LIN {X 0,Y 322.636,Z 898.882,A -85,B 0,C 180,E1 8627.078,E2 8627.078} C_VEL
LIN {X 0,Y 310.386,Z 918.046,A -85,B 0,C 180,E1 8625.849,E2 8625.849} C_VEL
LIN {X 0,Y 296.979,Z 936.905,A -85,B 0,C 180,E1 8624.35,E2 8624.35} C_VEL
LIN {X 0,Y 282.07,Z 955.374,A -85,B 0,C 180,E1 8622.47,E2 8622.47} C_VEL
LIN {X 0,Y 268.359,Z 970.812,A -85,B 0,C 180,E1 8620.504,E2 8620.504} C_VEL
LIN {X 0,Y 251.739,Z 987.693,A -85,B 0,C 180,E1 8617.738,E2 8617.738} C_VEL
LIN {X 0,Y 237.36,Z 1001.003,A -85,B 0,C 180,E1 8614.917,E2 8614.917} C_VEL
LIN {X 0,Y 219.956,Z 1015.757,A -85,B 0,C 180,E1 8610.786,E2 8610.786} C_VEL
LIN {X 0,Y 205.881,Z 1026.76,A -85,B 0,C 180,E1 8606.652,E2 8606.652} C_VEL
LIN {X 0,Y 190.594,Z 1038.003,A -85,B 0,C 180,E1 8600.935,E2 8600.935} C_VEL
LIN {X 0,Y 178.933,Z 1046.164,A -85,B 0,C 180,E1 8595.209,E2 8595.209} C_VEL
LIN {X 0,Y 167.932,Z 1053.856,A -85,B 0,C 180,E1 8587.827,E2 8587.827} C_VEL
LIN {X 0,Y 160.029,Z 1059.461,A -85,B 0,C 180,E1 8579.991,E2 8579.991} C_VEL
LIN {X 0,Y 154.899,Z 1063.661,A -85,B 0,C 180,E1 8571.589,E2 8571.589} C_VEL
LIN {X 0,Y 152.378,Z 1066.343,A -85,B 0,C 180,E1 8562.506,E2 8562.506} C_VEL
LIN {X 0,Y 151.995,Z 1067.325,A -85,B 0,C 180,E1 8555.663,E2 8555.663} C_VEL
LIN {X 0,Y 152.054,Z 1067.454,A -85,B 0,C 180,E1 8550,E2 8550} C_VEL
LIN {X 0,Y 151.999,Z 1066.865,A -85,B 0,C 180,E1 8543.958,E2 8543.958} C_VEL
LIN {X 0,Y 152.481,Z 1065.182,A -85,B 0,C 180,E1 8536.732,E2 8536.732} C_VEL
LIN {X 0,Y 154.529,Z 1062.318,A -85,B 0,C 180,E1 8529.153,E2 8529.153} C_VEL
LIN {X 0,Y 159.895,Z 1057.125,A -85,B 0,C 180,E1 8519.982,E2 8519.982} C_VEL
LIN {X 0,Y 167.312,Z 1050.928,A -85,B 0,C 180,E1 8512.441,E2 8512.441} C_VEL
LIN {X 0,Y 178.116,Z 1042.531,A -85,B 0,C 180,E1 8504.982,E2 8504.982} C_VEL
LIN {X 0,Y 190.201,Z 1032.991,A -85,B 0,C 180,E1 8498.919,E2 8498.919} C_VEL
LIN {X 0,Y 204.082,Z 1021.838,A -85,B 0,C 180,E1 8493.602,E2 8493.602} C_VEL
LIN {X 0,Y 218.709,Z 1009.161,A -85,B 0,C 180,E1 8489.166,E2 8489.166} C_VEL
LIN {X 0,Y 233.696,Z 995.401,A -85,B 0,C 180,E1 8485.474,E2 8485.474} C_VEL
LIN {X 0,Y 248.713,Z 980.22,A -85,B 0,C 180,E1 8482.383,E2 8482.383} C_VEL
LIN {X 0,Y 262.703,Z 964.888,A -85,B 0,C 180,E1 8479.928,E2 8479.928} C_VEL
LIN {X 0,Y 278.275,Z 945.943,A -85,B 0,C 180,E1 8477.567,E2 8477.567} C_VEL
LIN {X 0,Y 290.616,Z 929.27,A -85,B 0,C 180,E1 8475.92,E2 8475.92} C_VEL
LIN {X 0,Y 304.787,Z 907.829,A -85,B 0,C 180,E1 8474.244,E2 8474.244} C_VEL
LIN {X 0,Y 315.652,Z 889.153,A -85,B 0,C 180,E1 8473.081,E2 8473.081} C_VEL
LIN {X 0,Y 326.777,Z 867.511,A -85,B 0,C 180,E1 8471.993,E2 8471.993} C_VEL
LIN {X 0,Y 336.034,Z 846.319,A -85,B 0,C 180,E1 8471.152,E2 8471.152} C_VEL
LIN {X 0,Y 344.895,Z 822.678,A -85,B 0,C 180,E1 8470.416,E2 8470.416} C_VEL
LIN {X 0,Y 351.973,Z 798.939,A -85,B 0,C 180,E1 8469.86,E2 8469.86} C_VEL
LIN {X 0,Y 357.744,Z 774.619,A -85,B 0,C 180,E1 8469.413,E2 8469.413} C_VEL
LIN {X 0,Y 361.712,Z 750.039,A -85,B 0,C 180,E1 8469.033,E2 8469.033} C_VEL
LIN {X 0,Y 375.403,Z 627.088,A -85,B 0,C 180,E1 8467.345,E2 8467.345} C_VEL
LIN {X 0,Y 374.084,Z 623.885,A -85,B 0,C 180,E1 8465.368,E2 8465.368} C_VEL
LIN {X 0,Y 373.134,Z 621.334,A -85,B 0,C 180,E1 8463.38,E2 8463.38} C_VEL
LIN {X 0,Y 372.326,Z 618.216,A -85,B 0,C 180,E1 8458.615,E2 8458.615} C_VEL
LIN {X 0,Y 373.453,Z 622.113,A -85,B 0,C 180,E1 8453.466,E2 8453.466} C_VEL
LIN {X 0,Y 374.948,Z 625.93,A -85,B 0,C 180,E1 8450.87,E2 8450.87} C_VEL
LIN {X 0,Y 375.361,Z 627.187,A -85,B 0,C 180,E1 8450.268,E2 8450.268} C_VEL
LIN {X 0,Y 361.464,Z 750.862,A -85,B 0,C 180,E1 8448.59,E2 8448.59} C_VEL
LIN {X 0,Y 356.777,Z 777.011,A -85,B 0,C 180,E1 8448.155,E2 8448.155} C_VEL
LIN {X 0,Y 351.552,Z 798.416,A -85,B 0,C 180,E1 8447.699,E2 8447.699} C_VEL
LIN {X 0,Y 343.776,Z 823.534,A -85,B 0,C 180,E1 8446.998,E2 8446.998} C_VEL
LIN {X 0,Y 336.067,Z 843.934,A -85,B 0,C 180,E1 8446.27,E2 8446.27} C_VEL
LIN {X 0,Y 326.126,Z 866.42,A -85,B 0,C 180,E1 8445.275,E2 8445.275} C_VEL
LIN {X 0,Y 315.463,Z 886.892,A -85,B 0,C 180,E1 8444.148,E2 8444.148} C_VEL
LIN {X 0,Y 303.574,Z 907.129,A -85,B 0,C 180,E1 8442.781,E2 8442.781} C_VEL
LIN {X 0,Y 290.382,Z 926.631,A -85,B 0,C 180,E1 8441.114,E2 8441.114} C_VEL
LIN {X 0,Y 276.56,Z 945.065,A -85,B 0,C 180,E1 8439.163,E2 8439.163} C_VEL
LIN {X 0,Y 262.07,Z 962.147,A -85,B 0,C 180,E1 8436.853,E2 8436.853} C_VEL
LIN {X 0,Y 248.439,Z 976.868,A -85,B 0,C 180,E1 8434.36,E2 8434.36} C_VEL
LIN {X 0,Y 232.261,Z 992.697,A -85,B 0,C 180,E1 8430.891,E2 8430.891} C_VEL
LIN {X 0,Y 218.488,Z 1005.095,A -85,B 0,C 180,E1 8427.358,E2 8427.358} C_VEL
LIN {X 0,Y 202.958,Z 1018.013,A -85,B 0,C 180,E1 8422.484,E2 8422.484} C_VEL
LIN {X 0,Y 190.742,Z 1027.571,A -85,B 0,C 180,E1 8417.658,E2 8417.658} C_VEL
LIN {X 0,Y 177.939,Z 1037.213,A -85,B 0,C 180,E1 8411.106,E2 8411.106} C_VEL
LIN {X 0,Y 168.28,Z 1044.346,A -85,B 0,C 180,E1 8404.366,E2 8404.366} C_VEL
LIN {X 0,Y 160.311,Z 1050.558,A -85,B 0,C 180,E1 8396.285,E2 8396.285} C_VEL
LIN {X 0,Y 155.313,Z 1054.813,A -85,B 0,C 180,E1 8388,E2 8388} C_VEL
LIN {X 0,Y 152.896,Z 1057.51,A -85,B 0,C 180,E1 8380.17,E2 8380.17} C_VEL
LIN {X 0,Y 152.112,Z 1059.078,A -85,B 0,C 180,E1 8372.26,E2 8372.26} C_VEL
LIN {X 0,Y 152.062,Z 1059.433,A -85,B 0,C 180,E1 8365.474,E2 8365.474} C_VEL
LIN {X 0,Y 152.585,Z 1058.817,A -85,B 0,C 180,E1 8357.895,E2 8357.895} C_VEL
LIN {X 0,Y 154.442,Z 1057.168,A -85,B 0,C 180,E1 8350.327,E2 8350.327} C_VEL
LIN {X 0,Y 158.647,Z 1054.149,A -85,B 0,C 180,E1 8342.2,E2 8342.2} C_VEL
LIN {X 0,Y 166.393,Z 1048.96,A -85,B 0,C 180,E1 8333.494,E2 8333.494} C_VEL
LIN {X 0,Y 175.285,Z 1043.202,A -85,B 0,C 180,E1 8326.802,E2 8326.802} C_VEL
LIN {X 0,Y 188.413,Z 1034.522,A -85,B 0,C 180,E1 8319.691,E2 8319.691} C_VEL
LIN {X 0,Y 201.002,Z 1025.774,A -85,B 0,C 180,E1 8314.548,E2 8314.548} C_VEL
LIN {X 0,Y 216.974,Z 1013.934,A -85,B 0,C 180,E1 8309.428,E2 8309.428} C_VEL
LIN {X 0,Y 230.992,Z 1002.637,A -85,B 0,C 180,E1 8305.794,E2 8305.794} C_VEL
LIN {X 0,Y 246.815,Z 988.886,A -85,B 0,C 180,E1 8302.384,E2 8302.384} C_VEL
LIN {X 0,Y 262.135,Z 974.029,A -85,B 0,C 180,E1 8299.583,E2 8299.583} C_VEL
LIN {X 0,Y 277.791,Z 957.455,A -85,B 0,C 180,E1 8297.128,E2 8297.128} C_VEL
LIN {X 0,Y 292.122,Z 940.304,A -85,B 0,C 180,E1 8295.15,E2 8295.15} C_VEL
LIN {X 0,Y 305.426,Z 922.738,A -85,B 0,C 180,E1 8293.515,E2 8293.515} C_VEL
LIN {X 0,Y 318.945,Z 902.467,A -85,B 0,C 180,E1 8292.008,E2 8292.008} C_VEL
LIN {X 0,Y 329.913,Z 883.896,A -85,B 0,C 180,E1 8290.897,E2 8290.897} C_VEL
LIN {X 0,Y 341.912,Z 860.439,A -85,B 0,C 180,E1 8289.76,E2 8289.76} C_VEL
LIN {X 0,Y 350.295,Z 841.325,A -85,B 0,C 180,E1 8289.021,E2 8289.021} C_VEL
LIN {X 0,Y 358.98,Z 818.103,A -85,B 0,C 180,E1 8288.288,E2 8288.288} C_VEL
LIN {X 0,Y 365.752,Z 795.493,A -85,B 0,C 180,E1 8287.729,E2 8287.729} C_VEL
LIN {X 0,Y 371.547,Z 771.253,A -85,B 0,C 180,E1 8287.27,E2 8287.27} C_VEL
LIN {X 0,Y 375.564,Z 746.851,A -85,B 0,C 180,E1 8286.912,E2 8286.912} C_VEL
LIN {X 0,Y 388.046,Z 637.82,A -85,B 0,C 180,E1 8285.471,E2 8285.471} C_VEL
LIN {X 0,Y 387.076,Z 635.217,A -85,B 0,C 180,E1 8283.406,E2 8283.406} C_VEL
LIN {X 0,Y 386.369,Z 632.327,A -85,B 0,C 180,E1 8279.11,E2 8279.11} C_VEL
LIN {X 0,Y 387.338,Z 635.859,A -85,B 0,C 180,E1 8274.296,E2 8274.296} C_VEL
LIN {X 0,Y 388.067,Z 638.147,A -85,B 0,C 180,E1 8272.782,E2 8272.782} C_VEL
LIN {X 0,Y 374.709,Z 754.049,A -85,B 0,C 180,E1 8271.265,E2 8271.265} C_VEL
LIN {X 0,Y 372.793,Z 765.718,A -85,B 0,C 180,E1 8271.095,E2 8271.095} C_VEL
LIN {X 0,Y 371.277,Z 773.315,A -85,B 0,C 180,E1 8271.153,E2 8271.153} C_VEL
LIN {X 0,Y 365.77,Z 793.42,A -85,B 0,C 180,E1 8271.797,E2 8271.797} C_VEL
LIN {X 0,Y 363.895,Z 799.825,A -85,B 0,C 180,E1 8271.782,E2 8271.782} C_VEL
LIN {X 0,Y 356.423,Z 823.805,A -85,B 0,C 180,E1 8271.287,E2 8271.287} C_VEL
LIN {X 0,Y 348.041,Z 845.479,A -85,B 0,C 180,E1 8270.695,E2 8270.695} C_VEL
LIN {X 0,Y 338.627,Z 866.422,A -85,B 0,C 180,E1 8269.98,E2 8269.98} C_VEL
LIN {X 0,Y 326.946,Z 888.501,A -85,B 0,C 180,E1 8269.023,E2 8269.023} C_VEL
LIN {X 0,Y 315.383,Z 907.692,A -85,B 0,C 180,E1 8267.978,E2 8267.978} C_VEL
LIN {X 0,Y 300.755,Z 928.939,A -85,B 0,C 180,E1 8266.519,E2 8266.519} C_VEL
LIN {X 0,Y 287.707,Z 945.803,A -85,B 0,C 180,E1 8265.05,E2 8265.05} C_VEL
LIN {X 0,Y 270.941,Z 965.149,A -85,B 0,C 180,E1 8262.906,E2 8262.906} C_VEL
LIN {X 0,Y 256.316,Z 980.279,A -85,B 0,C 180,E1 8260.742,E2 8260.742} C_VEL
LIN {X 0,Y 238.838,Z 996.651,A -85,B 0,C 180,E1 8257.7,E2 8257.7} C_VEL
LIN {X 0,Y 223.7,Z 1009.49,A -85,B 0,C 180,E1 8254.541,E2 8254.541} C_VEL
LIN {X 0,Y 207.161,Z 1022.449,A -85,B 0,C 180,E1 8250.319,E2 8250.319} C_VEL
LIN {X 0,Y 192.57,Z 1032.93,A -85,B 0,C 180,E1 8245.648,E2 8245.648} C_VEL
LIN {X 0,Y 178.251,Z 1042.757,A -85,B 0,C 180,E1 8239.719,E2 8239.719} C_VEL
LIN {X 0,Y 166.033,Z 1050.649,A -85,B 0,C 180,E1 8232.884,E2 8232.884} C_VEL
LIN {X 0,Y 156.312,Z 1057.058,A -85,B 0,C 180,E1 8225.149,E2 8225.149} C_VEL
LIN {X 0,Y 148.961,Z 1062.123,A -85,B 0,C 180,E1 8215.912,E2 8215.912} C_VEL
LIN {X 0,Y 145.407,Z 1065.091,A -85,B 0,C 180,E1 8207.612,E2 8207.612} C_VEL
LIN {X 0,Y 144.033,Z 1066.956,A -85,B 0,C 180,E1 8198.383,E2 8198.383} C_VEL
LIN {X 0,Y 144.033,Z 1067.319,A -85,B 0,C 180,E1 8191.482,E2 8191.482} C_VEL
LIN {X 0,Y 144.001,Z 1066.922,A -85,B 0,C 180,E1 8185.22,E2 8185.22} C_VEL
LIN {X 0,Y 144.399,Z 1065.305,A -85,B 0,C 180,E1 8177.198,E2 8177.198} C_VEL
LIN {X 0,Y 146.424,Z 1062.574,A -85,B 0,C 180,E1 8169.201,E2 8169.201} C_VEL
LIN {X 0,Y 151.07,Z 1058.295,A -85,B 0,C 180,E1 8160.674,E2 8160.674} C_VEL
LIN {X 0,Y 159.581,Z 1051.598,A -85,B 0,C 180,E1 8151.662,E2 8151.662} C_VEL
LIN {X 0,Y 169.211,Z 1044.499,A -85,B 0,C 180,E1 8144.839,E2 8144.839} C_VEL
LIN {X 0,Y 183.245,Z 1034.109,A -85,B 0,C 180,E1 8137.702,E2 8137.702} C_VEL
LIN {X 0,Y 196.167,Z 1024.178,A -85,B 0,C 180,E1 8132.751,E2 8132.751} C_VEL
LIN {X 0,Y 213.075,Z 1010.331,A -85,B 0,C 180,E1 8127.683,E2 8127.683} C_VEL
LIN {X 0,Y 227.093,Z 997.928,A -85,B 0,C 180,E1 8124.298,E2 8124.298} C_VEL
LIN {X 0,Y 244.223,Z 981.397,A -85,B 0,C 180,E1 8120.867,E2 8120.867} C_VEL
LIN {X 0,Y 258.302,Z 966.413,A -85,B 0,C 180,E1 8118.487,E2 8118.487} C_VEL
LIN {X 0,Y 273.869,Z 948.18,A -85,B 0,C 180,E1 8116.218,E2 8116.218} C_VEL
LIN {X 0,Y 287.136,Z 930.725,A -85,B 0,C 180,E1 8114.516,E2 8114.516} C_VEL
LIN {X 0,Y 300.657,Z 911.038,A -85,B 0,C 180,E1 8112.986,E2 8112.986} C_VEL
LIN {X 0,Y 312.993,Z 890.336,A -85,B 0,C 180,E1 8111.722,E2 8111.722} C_VEL
LIN {X 0,Y 323.623,Z 870.228,A -85,B 0,C 180,E1 8110.73,E2 8110.73} C_VEL
LIN {X 0,Y 333.881,Z 847.437,A -85,B 0,C 180,E1 8109.846,E2 8109.846} C_VEL
LIN {X 0,Y 341.873,Z 826.674,A -85,B 0,C 180,E1 8109.214,E2 8109.214} C_VEL
LIN {X 0,Y 349.827,Z 801.391,A -85,B 0,C 180,E1 8108.625,E2 8108.625} C_VEL
LIN {X 0,Y 355.241,Z 779.522,A -85,B 0,C 180,E1 8108.229,E2 8108.229} C_VEL
LIN {X 0,Y 360.011,Z 752.727,A -85,B 0,C 180,E1 8107.817,E2 8107.817} C_VEL
LIN {X 0,Y 373.612,Z 633.289,A -85,B 0,C 180,E1 8106.23,E2 8106.23} C_VEL
LIN {X 0,Y 372.089,Z 629.213,A -85,B 0,C 180,E1 8103.235,E2 8103.235} C_VEL
LIN {X 0,Y 371.346,Z 626.202,A -85,B 0,C 180,E1 8098.611,E2 8098.611} C_VEL
LIN {X 0,Y 372.364,Z 629.922,A -85,B 0,C 180,E1 8093.679,E2 8093.679} C_VEL
LIN {X 0,Y 373.577,Z 633.217,A -85,B 0,C 180,E1 8091.404,E2 8091.404} C_VEL
LIN {X 0,Y 360.091,Z 751.213,A -85,B 0,C 180,E1 8089.84,E2 8089.84} C_VEL
LIN {X 0,Y 355.373,Z 777.18,A -85,B 0,C 180,E1 8089.424,E2 8089.424} C_VEL
LIN {X 0,Y 350.07,Z 798.648,A -85,B 0,C 180,E1 8088.985,E2 8088.985} C_VEL
LIN {X 0,Y 342.069,Z 824.119,A -85,B 0,C 180,E1 8088.301,E2 8088.301} C_VEL
LIN {X 0,Y 334.26,Z 844.475,A -85,B 0,C 180,E1 8087.601,E2 8087.601} C_VEL
LIN {X 0,Y 324.182,Z 866.895,A -85,B 0,C 180,E1 8086.645,E2 8086.645} C_VEL
LIN {X 0,Y 313.817,Z 886.539,A -85,B 0,C 180,E1 8085.606,E2 8085.606} C_VEL
LIN {X 0,Y 301.733,Z 906.842,A -85,B 0,C 180,E1 8084.294,E2 8084.294} C_VEL
LIN {X 0,Y 288.501,Z 926.158,A -85,B 0,C 180,E1 8082.713,E2 8082.713} C_VEL
LIN {X 0,Y 275.499,Z 943.251,A -85,B 0,C 180,E1 8080.988,E2 8080.988} C_VEL
LIN {X 0,Y 259.827,Z 961.586,A -85,B 0,C 180,E1 8078.636,E2 8078.636} C_VEL
LIN {X 0,Y 245.843,Z 976.377,A -85,B 0,C 180,E1 8076.222,E2 8076.222} C_VEL
LIN {X 0,Y 229.224,Z 992.292,A -85,B 0,C 180,E1 8072.855,E2 8072.855} C_VEL
LIN {X 0,Y 215.661,Z 1004.157,A -85,B 0,C 180,E1 8069.583,E2 8069.583} C_VEL
LIN {X 0,Y 200.122,Z 1016.792,A -85,B 0,C 180,E1 8065.026,E2 8065.026} C_VEL
LIN {X 0,Y 186.559,Z 1026.959,A -85,B 0,C 180,E1 8060.034,E2 8060.034} C_VEL
LIN {X 0,Y 173.444,Z 1036.446,A -85,B 0,C 180,E1 8053.772,E2 8053.772} C_VEL
LIN {X 0,Y 162.464,Z 1044.017,A -85,B 0,C 180,E1 8046.654,E2 8046.654} C_VEL
LIN {X 0,Y 153.982,Z 1050.121,A -85,B 0,C 180,E1 8038.72,E2 8038.72} C_VEL
LIN {X 0,Y 148.005,Z 1054.743,A -85,B 0,C 180,E1 8029.742,E2 8029.742} C_VEL
LIN {X 0,Y 145.243,Z 1057.412,A -85,B 0,C 180,E1 8021.919,E2 8021.919} C_VEL
LIN {X 0,Y 144.199,Z 1058.976,A -85,B 0,C 180,E1 8014.374,E2 8014.374} C_VEL
LIN {X 0,Y 144.037,Z 1059.569,A -85,B 0,C 180,E1 8007.613,E2 8007.613} C_VEL
LIN {X 0,Y 144.314,Z 1059.398,A -85,B 0,C 180,E1 8000.428,E2 8000.428} C_VEL
LIN {X 0,Y 146.072,Z 1057.914,A -85,B 0,C 180,E1 7991.233,E2 7991.233} C_VEL
LIN {X 0,Y 149.888,Z 1055.271,A -85,B 0,C 180,E1 7983.024,E2 7983.024} C_VEL
LIN {X 0,Y 156.774,Z 1051.046,A -85,B 0,C 180,E1 7974.522,E2 7974.522} C_VEL
LIN {X 0,Y 166.876,Z 1044.865,A -85,B 0,C 180,E1 7966.444,E2 7966.444} C_VEL
LIN {X 0,Y 177.931,Z 1038.053,A -85,B 0,C 180,E1 7960.159,E2 7960.159} C_VEL
LIN {X 0,Y 192.704,Z 1028.454,A -85,B 0,C 180,E1 7953.881,E2 7953.881} C_VEL
LIN {X 0,Y 206.466,Z 1018.863,A -85,B 0,C 180,E1 7949.341,E2 7949.341} C_VEL
LIN {X 0,Y 223.283,Z 1006.192,A -85,B 0,C 180,E1 7944.894,E2 7944.894} C_VEL
LIN {X 0,Y 238.041,Z 993.951,A -85,B 0,C 180,E1 7941.694,E2 7941.694} C_VEL
LIN {X 0,Y 254.411,Z 979.174,A -85,B 0,C 180,E1 7938.705,E2 7938.705} C_VEL
LIN {X 0,Y 269.808,Z 963.547,A -85,B 0,C 180,E1 7936.294,E2 7936.294} C_VEL
LIN {X 0,Y 285.132,Z 946.472,A -85,B 0,C 180,E1 7934.21,E2 7934.21} C_VEL
LIN {X 0,Y 299.537,Z 928.245,A -85,B 0,C 180,E1 7932.472,E2 7932.472} C_VEL
LIN {X 0,Y 312.45,Z 910.056,A -85,B 0,C 180,E1 7931.07,E2 7931.07} C_VEL
LIN {X 0,Y 325.685,Z 888.747,A -85,B 0,C 180,E1 7929.767,E2 7929.767} C_VEL
LIN {X 0,Y 335.946,Z 869.895,A -85,B 0,C 180,E1 7928.831,E2 7928.831} C_VEL
LIN {X 0,Y 346.945,Z 846.423,A -85,B 0,C 180,E1 7927.888,E2 7927.888} C_VEL
LIN {X 0,Y 354.795,Z 826.568,A -85,B 0,C 180,E1 7927.247,E2 7927.247} C_VEL
LIN {X 0,Y 362.673,Z 802.827,A -85,B 0,C 180,E1 7926.638,E2 7926.638} C_VEL
LIN {X 0,Y 368.63,Z 779.656,A -85,B 0,C 180,E1 7926.185,E2 7926.185} C_VEL
LIN {X 0,Y 373.408,Z 755.336,A -85,B 0,C 180,E1 7925.81,E2 7925.81} C_VEL
LIN {X 0,Y 379.555,Z 704.728,A -85,B 0,C 180,E1 7925.156,E2 7925.156} C_VEL
LIN {X 0,Y 386.488,Z 644.435,A -85,B 0,C 180,E1 7924.385,E2 7924.385} C_VEL
LIN {X 0,Y 385.979,Z 642.999,A -85,B 0,C 180,E1 7923.119,E2 7923.119} C_VEL
LIN {X 0,Y 385.387,Z 640.321,A -85,B 0,C 180,E1 7919.108,E2 7919.108} C_VEL
LIN {X 0,Y 386.259,Z 643.666,A -85,B 0,C 180,E1 7914.504,E2 7914.504} C_VEL
LIN {X 0,Y 386.489,Z 644.784,A -85,B 0,C 180,E1 7913.879,E2 7913.879} C_VEL
LIN {X 0,Y 373.686,Z 754.037,A -85,B 0,C 180,E1 7912.483,E2 7912.483} C_VEL
LIN {X 0,Y 368.824,Z 780.191,A -85,B 0,C 180,E1 7912.104,E2 7912.104} C_VEL
LIN {X 0,Y 363.895,Z 799.825,A -85,B 0,C 180,E1 7911.782,E2 7911.782} C_VEL
LIN {X 0,Y 361.669,Z 807.26,A -85,B 0,C 180,E1 7911.819,E2 7911.819} C_VEL
LIN {X 0,Y 354.68,Z 825.951,A -85,B 0,C 180,E1 7912.365,E2 7912.365} C_VEL
LIN {X 0,Y 351.901,Z 833.042,A -85,B 0,C 180,E1 7912.345,E2 7912.345} C_VEL
LIN {X 0,Y 341.59,Z 857.457,A -85,B 0,C 180,E1 7911.643,E2 7911.643} C_VEL
LIN {X 0,Y 331.506,Z 877.698,A -85,B 0,C 180,E1 7910.894,E2 7910.894} C_VEL
LIN {X 0,Y 318.47,Z 900.334,A -85,B 0,C 180,E1 7909.829,E2 7909.829} C_VEL
LIN {X 0,Y 306.359,Z 918.658,A -85,B 0,C 180,E1 7908.744,E2 7908.744} C_VEL
LIN {X 0,Y 292.091,Z 937.956,A -85,B 0,C 180,E1 7907.321,E2 7907.321} C_VEL
LIN {X 0,Y 277.137,Z 955.733,A -85,B 0,C 180,E1 7905.634,E2 7905.634} C_VEL
LIN {X 0,Y 260.71,Z 973.388,A -85,B 0,C 180,E1 7903.499,E2 7903.499} C_VEL
LIN {X 0,Y 244.275,Z 989.022,A -85,B 0,C 180,E1 7901.006,E2 7901.006} C_VEL
LIN {X 0,Y 227.573,Z 1003.58,A -85,B 0,C 180,E1 7897.983,E2 7897.983} C_VEL
LIN {X 0,Y 210.824,Z 1016.635,A -85,B 0,C 180,E1 7894.306,E2 7894.306} C_VEL
LIN {X 0,Y 195.09,Z 1028.025,A -85,B 0,C 180,E1 7890.017,E2 7890.017} C_VEL
LIN {X 0,Y 179.302,Z 1038.497,A -85,B 0,C 180,E1 7884.506,E2 7884.506} C_VEL
LIN {X 0,Y 166.53,Z 1046.54,A -85,B 0,C 180,E1 7878.637,E2 7878.637} C_VEL
LIN {X 0,Y 153.385,Z 1054.528,A -85,B 0,C 180,E1 7870.193,E2 7870.193} C_VEL
LIN {X 0,Y 145.319,Z 1059.505,A -85,B 0,C 180,E1 7862.459,E2 7862.459} C_VEL
LIN {X 0,Y 139.028,Z 1063.816,A -85,B 0,C 180,E1 7852.407,E2 7852.407} C_VEL
LIN {X 0,Y 136.508,Z 1066.001,A -85,B 0,C 180,E1 7843.556,E2 7843.556} C_VEL
LIN {X 0,Y 135.999,Z 1066.928,A -85,B 0,C 180,E1 7835.908,E2 7835.908} C_VEL
LIN {X 0,Y 136.059,Z 1067.021,A -85,B 0,C 180,E1 7830,E2 7830} C_VEL
LIN {X 0,Y 136.006,Z 1066.417,A -85,B 0,C 180,E1 7823.245,E2 7823.245} C_VEL
LIN {X 0,Y 136.711,Z 1064.717,A -85,B 0,C 180,E1 7815.168,E2 7815.168} C_VEL
LIN {X 0,Y 139.354,Z 1061.814,A -85,B 0,C 180,E1 7806.698,E2 7806.698} C_VEL
LIN {X 0,Y 145.833,Z 1056.613,A -85,B 0,C 180,E1 7796.735,E2 7796.735} C_VEL
LIN {X 0,Y 154.501,Z 1050.4,A -85,B 0,C 180,E1 7788.691,E2 7788.691} C_VEL
LIN {X 0,Y 166.227,Z 1042.388,A -85,B 0,C 180,E1 7781.245,E2 7781.245} C_VEL
LIN {X 0,Y 179.96,Z 1032.608,A -85,B 0,C 180,E1 7774.91,E2 7774.91} C_VEL
LIN {X 0,Y 195.382,Z 1021.235,A -85,B 0,C 180,E1 7769.542,E2 7769.542} C_VEL
LIN {X 0,Y 211.129,Z 1008.531,A -85,B 0,C 180,E1 7765.229,E2 7765.229} C_VEL
LIN {X 0,Y 227.067,Z 994.761,A -85,B 0,C 180,E1 7761.699,E2 7761.699} C_VEL
LIN {X 0,Y 243.473,Z 978.966,A -85,B 0,C 180,E1 7758.683,E2 7758.683} C_VEL
LIN {X 0,Y 258.429,Z 963.247,A -85,B 0,C 180,E1 7756.355,E2 7756.355} C_VEL
LIN {X 0,Y 273.92,Z 944.994,A -85,B 0,C 180,E1 7754.268,E2 7754.268} C_VEL
LIN {X 0,Y 287.009,Z 927.872,A -85,B 0,C 180,E1 7752.717,E2 7752.717} C_VEL
LIN {X 0,Y 301.23,Z 906.903,A -85,B 0,C 180,E1 7751.225,E2 7751.225} C_VEL
LIN {X 0,Y 312.372,Z 888.252,A -85,B 0,C 180,E1 7750.168,E2 7750.168} C_VEL
LIN {X 0,Y 324.093,Z 865.864,A -85,B 0,C 180,E1 7749.155,E2 7749.155} C_VEL
LIN {X 0,Y 333.067,Z 845.762,A -85,B 0,C 180,E1 7748.436,E2 7748.436} C_VEL
LIN {X 0,Y 341.865,Z 822.855,A -85,B 0,C 180,E1 7747.787,E2 7747.787} C_VEL
LIN {X 0,Y 349.212,Z 798.836,A -85,B 0,C 180,E1 7747.277,E2 7747.277} C_VEL
LIN {X 0,Y 355.105,Z 774.615,A -85,B 0,C 180,E1 7746.871,E2 7746.871} C_VEL
LIN {X 0,Y 359.227,Z 749.857,A -85,B 0,C 180,E1 7746.514,E2 7746.514} C_VEL
LIN {X 0,Y 371.93,Z 639.67,A -85,B 0,C 180,E1 7745.09,E2 7745.09} C_VEL
LIN {X 0,Y 370.985,Z 636.993,A -85,B 0,C 180,E1 7742.935,E2 7742.935} C_VEL
LIN {X 0,Y 370.365,Z 634.188,A -85,B 0,C 180,E1 7738.608,E2 7738.608} C_VEL
LIN {X 0,Y 371.309,Z 637.843,A -85,B 0,C 180,E1 7733.816,E2 7733.816} C_VEL
LIN {X 0,Y 371.884,Z 639.748,A -85,B 0,C 180,E1 7732.543,E2 7732.543} C_VEL
LIN {X 0,Y 358.891,Z 751.554,A -85,B 0,C 180,E1 7731.1,E2 7731.1} C_VEL
LIN {X 0,Y 354.116,Z 777.471,A -85,B 0,C 180,E1 7730.7,E2 7730.7} C_VEL
LIN {X 0,Y 348.715,Z 799.063,A -85,B 0,C 180,E1 7730.277,E2 7730.277} C_VEL
LIN {X 0,Y 340.54,Z 824.701,A -85,B 0,C 180,E1 7729.616,E2 7729.616} C_VEL
LIN {X 0,Y 332.636,Z 845.015,A -85,B 0,C 180,E1 7728.945,E2 7728.945} C_VEL
LIN {X 0,Y 322.011,Z 868.172,A -85,B 0,C 180,E1 7727.992,E2 7727.992} C_VEL
LIN {X 0,Y 311.508,Z 887.711,A -85,B 0,C 180,E1 7726.993,E2 7726.993} C_VEL
LIN {X 0,Y 299.205,Z 907.957,A -85,B 0,C 180,E1 7725.726,E2 7725.726} C_VEL
LIN {X 0,Y 285.765,Z 927.152,A -85,B 0,C 180,E1 7724.201,E2 7724.201} C_VEL
LIN {X 0,Y 271.231,Z 945.815,A -85,B 0,C 180,E1 7722.355,E2 7722.355} C_VEL
LIN {X 0,Y 256.135,Z 962.851,A -85,B 0,C 180,E1 7720.187,E2 7720.187} C_VEL
LIN {X 0,Y 241.033,Z 978.385,A -85,B 0,C 180,E1 7717.681,E2 7717.681} C_VEL
LIN {X 0,Y 224.836,Z 993.303,A -85,B 0,C 180,E1 7714.526,E2 7714.526} C_VEL
LIN {X 0,Y 210.146,Z 1005.718,A -85,B 0,C 180,E1 7711.102,E2 7711.102} C_VEL
LIN {X 0,Y 193.459,Z 1018.601,A -85,B 0,C 180,E1 7706.318,E2 7706.318} C_VEL
LIN {X 0,Y 180.153,Z 1028.144,A -85,B 0,C 180,E1 7701.498,E2 7701.498} C_VEL
LIN {X 0,Y 165.451,Z 1038.099,A -85,B 0,C 180,E1 7694.51,E2 7694.51} C_VEL
LIN {X 0,Y 155.106,Z 1044.871,A -85,B 0,C 180,E1 7687.764,E2 7687.764} C_VEL
LIN {X 0,Y 145.923,Z 1051.053,A -85,B 0,C 180,E1 7679.111,E2 7679.111} C_VEL
LIN {X 0,Y 140.019,Z 1055.292,A -85,B 0,C 180,E1 7670.046,E2 7670.046} C_VEL
LIN {X 0,Y 137.097,Z 1057.973,A -85,B 0,C 180,E1 7661.357,E2 7661.357} C_VEL
LIN {X 0,Y 136.125,Z 1059.517,A -85,B 0,C 180,E1 7652.526,E2 7652.526} C_VEL
LIN {X 0,Y 136.078,Z 1059.854,A -85,B 0,C 180,E1 7644.941,E2 7644.941} C_VEL
LIN {X 0,Y 136.713,Z 1059.293,A -85,B 0,C 180,E1 7636.895,E2 7636.895} C_VEL
LIN {X 0,Y 138.991,Z 1057.679,A -85,B 0,C 180,E1 7628.476,E2 7628.476} C_VEL
LIN {X 0,Y 143.709,Z 1054.848,A -85,B 0,C 180,E1 7619.937,E2 7619.937} C_VEL
LIN {X 0,Y 152.977,Z 1049.573,A -85,B 0,C 180,E1 7610.167,E2 7610.167} C_VEL
LIN {X 0,Y 163.062,Z 1043.85,A -85,B 0,C 180,E1 7603.138,E2 7603.138} C_VEL
LIN {X 0,Y 177.76,Z 1035.167,A -85,B 0,C 180,E1 7595.803,E2 7595.803} C_VEL
LIN {X 0,Y 191.676,Z 1026.338,A -85,B 0,C 180,E1 7590.601,E2 7590.601} C_VEL
LIN {X 0,Y 208.569,Z 1014.772,A -85,B 0,C 180,E1 7585.673,E2 7585.673} C_VEL
LIN {X 0,Y 224.273,Z 1002.903,A -85,B 0,C 180,E1 7581.994,E2 7581.994} C_VEL
LIN {X 0,Y 240.811,Z 989.282,A -85,B 0,C 180,E1 7578.792,E2 7578.792} C_VEL
LIN {X 0,Y 256.218,Z 975.058,A -85,B 0,C 180,E1 7576.257,E2 7576.257} C_VEL
LIN {X 0,Y 271.177,Z 959.936,A -85,B 0,C 180,E1 7574.131,E2 7574.131} C_VEL
LIN {X 0,Y 286.867,Z 942.134,A -85,B 0,C 180,E1 7572.174,E2 7572.174} C_VEL
LIN {X 0,Y 299.674,Z 925.914,A -85,B 0,C 180,E1 7570.747,E2 7570.747} C_VEL
LIN {X 0,Y 314.092,Z 905.408,A -85,B 0,C 180,E1 7569.298,E2 7569.298} C_VEL
LIN {X 0,Y 325.346,Z 887.102,A -85,B 0,C 180,E1 7568.268,E2 7568.268} C_VEL
LIN {X 0,Y 336.695,Z 866.245,A -85,B 0,C 180,E1 7567.303,E2 7567.303} C_VEL
LIN {X 0,Y 346.692,Z 844.499,A -85,B 0,C 180,E1 7566.502,E2 7566.502} C_VEL
LIN {X 0,Y 354.828,Z 823.837,A -85,B 0,C 180,E1 7565.88,E2 7565.88} C_VEL
LIN {X 0,Y 362.88,Z 798.729,A -85,B 0,C 180,E1 7565.289,E2 7565.289} C_VEL
LIN {X 0,Y 368.398,Z 776.886,A -85,B 0,C 180,E1 7564.897,E2 7564.897} C_VEL
LIN {X 0,Y 373.276,Z 750.254,A -85,B 0,C 180,E1 7564.519,E2 7564.519} C_VEL
LIN {X 0,Y 385.06,Z 651.072,A -85,B 0,C 180,E1 7563.275,E2 7563.275} C_VEL
LIN {X 0,Y 384.406,Z 648.313,A -85,B 0,C 180,E1 7559.106,E2 7559.106} C_VEL
LIN {X 0,Y 385.072,Z 651.262,A -85,B 0,C 180,E1 7554.986,E2 7554.986} C_VEL
LIN {X 0,Y 372.858,Z 753.848,A -85,B 0,C 180,E1 7553.71,E2 7553.71} C_VEL
LIN {X 0,Y 367.945,Z 779.984,A -85,B 0,C 180,E1 7553.346,E2 7553.346} C_VEL
LIN {X 0,Y 362.317,Z 801.977,A -85,B 0,C 180,E1 7553,E2 7553} C_VEL
LIN {X 0,Y 354.003,Z 827.41,A -85,B 0,C 180,E1 7552.484,E2 7552.484} C_VEL
LIN {X 0,Y 351.901,Z 833.042,A -85,B 0,C 180,E1 7552.345,E2 7552.345} C_VEL
LIN {X 0,Y 348.961,Z 840.282,A -85,B 0,C 180,E1 7552.318,E2 7552.318} C_VEL
LIN {X 0,Y 340.298,Z 858.245,A -85,B 0,C 180,E1 7552.791,E2 7552.791} C_VEL
LIN {X 0,Y 336.89,Z 865.112,A -85,B 0,C 180,E1 7552.734,E2 7552.734} C_VEL
LIN {X 0,Y 325.209,Z 886.908,A -85,B 0,C 180,E1 7551.9,E2 7551.9} C_VEL
LIN {X 0,Y 313.827,Z 905.472,A -85,B 0,C 180,E1 7551.003,E2 7551.003} C_VEL
LIN {X 0,Y 299.256,Z 926.414,A -85,B 0,C 180,E1 7549.736,E2 7549.736} C_VEL
LIN {X 0,Y 285.785,Z 943.458,A -85,B 0,C 180,E1 7548.421,E2 7548.421} C_VEL
LIN {X 0,Y 270.221,Z 961.244,A -85,B 0,C 180,E1 7546.697,E2 7546.697} C_VEL
LIN {X 0,Y 254.044,Z 977.534,A -85,B 0,C 180,E1 7544.643,E2 7544.643} C_VEL
LIN {X 0,Y 238.257,Z 992.011,A -85,B 0,C 180,E1 7542.297,E2 7542.297} C_VEL
LIN {X 0,Y 220.432,Z 1006.67,A -85,B 0,C 180,E1 7539.136,E2 7539.136} C_VEL
LIN {X 0,Y 204.985,Z 1018.231,A -85,B 0,C 180,E1 7535.806,E2 7535.806} C_VEL
LIN {X 0,Y 186.511,Z 1030.839,A -85,B 0,C 180,E1 7530.8,E2 7530.8} C_VEL
LIN {X 0,Y 171.931,Z 1039.978,A -85,B 0,C 180,E1 7525.672,E2 7525.672} C_VEL
LIN {X 0,Y 156.524,Z 1049.055,A -85,B 0,C 180,E1 7518.366,E2 7518.366} C_VEL
LIN {X 0,Y 145.248,Z 1055.417,A -85,B 0,C 180,E1 7510.778,E2 7510.778} C_VEL
LIN {X 0,Y 135.786,Z 1060.915,A -85,B 0,C 180,E1 7501.028,E2 7501.028} C_VEL
LIN {X 0,Y 130.572,Z 1064.21,A -85,B 0,C 180,E1 7491.566,E2 7491.566} C_VEL
LIN {X 0,Y 128.359,Z 1066.085,A -85,B 0,C 180,E1 7482.598,E2 7482.598} C_VEL
LIN {X 0,Y 128.002,Z 1066.818,A -85,B 0,C 180,E1 7474.48,E2 7474.48} C_VEL
LIN {X 0,Y 128.037,Z 1066.713,A -85,B 0,C 180,E1 7468.21,E2 7468.21} C_VEL
LIN {X 0,Y 128.044,Z 1065.979,A -85,B 0,C 180,E1 7461.468,E2 7461.468} C_VEL
LIN {X 0,Y 129.155,Z 1064.128,A -85,B 0,C 180,E1 7452.891,E2 7452.891} C_VEL
LIN {X 0,Y 133.454,Z 1060.36,A -85,B 0,C 180,E1 7442.32,E2 7442.32} C_VEL
LIN {X 0,Y 140.894,Z 1055.047,A -85,B 0,C 180,E1 7432.899,E2 7432.899} C_VEL
LIN {X 0,Y 151.918,Z 1047.938,A -85,B 0,C 180,E1 7424.159,E2 7424.159} C_VEL
LIN {X 0,Y 165.139,Z 1039.209,A -85,B 0,C 180,E1 7416.943,E2 7416.943} C_VEL
LIN {X 0,Y 179.785,Z 1029.321,A -85,B 0,C 180,E1 7411.076,E2 7411.076} C_VEL
LIN {X 0,Y 195.964,Z 1017.429,A -85,B 0,C 180,E1 7406.101,E2 7406.101} C_VEL
LIN {X 0,Y 211.756,Z 1004.997,A -85,B 0,C 180,E1 7402.257,E2 7402.257} C_VEL
LIN {X 0,Y 228.856,Z 990.097,A -85,B 0,C 180,E1 7398.863,E2 7398.863} C_VEL
LIN {X 0,Y 243.866,Z 975.771,A -85,B 0,C 180,E1 7396.375,E2 7396.375} C_VEL
LIN {X 0,Y 260.896,Z 957.673,A -85,B 0,C 180,E1 7393.972,E2 7393.972} C_VEL
LIN {X 0,Y 274.295,Z 941.809,A -85,B 0,C 180,E1 7392.328,E2 7392.328} C_VEL
LIN {X 0,Y 289.489,Z 921.719,A -85,B 0,C 180,E1 7390.687,E2 7390.687} C_VEL
LIN {X 0,Y 302.091,Z 902.766,A -85,B 0,C 180,E1 7389.478,E2 7389.478} C_VEL
LIN {X 0,Y 314.82,Z 881.085,A -85,B 0,C 180,E1 7388.372,E2 7388.372} C_VEL
LIN {X 0,Y 325.281,Z 860.292,A -85,B 0,C 180,E1 7387.546,E2 7387.546} C_VEL
LIN {X 0,Y 334.799,Z 838.531,A -85,B 0,C 180,E1 7386.861,E2 7386.861} C_VEL
LIN {X 0,Y 343.033,Z 815.564,A -85,B 0,C 180,E1 7386.299,E2 7386.299} C_VEL
LIN {X 0,Y 349.627,Z 793.272,A -85,B 0,C 180,E1 7385.877,E2 7385.877} C_VEL
LIN {X 0,Y 355.299,Z 767.873,A -85,B 0,C 180,E1 7385.491,E2 7385.491} C_VEL
LIN {X 0,Y 358.865,Z 745.266,A -85,B 0,C 180,E1 7385.182,E2 7385.182} C_VEL
LIN {X 0,Y 370.36,Z 646.203,A -85,B 0,C 180,E1 7383.909,E2 7383.909} C_VEL
LIN {X 0,Y 369.892,Z 644.775,A -85,B 0,C 180,E1 7382.634,E2 7382.634} C_VEL
LIN {X 0,Y 369.384,Z 642.181,A -85,B 0,C 180,E1 7378.604,E2 7378.604} C_VEL
LIN {X 0,Y 370.228,Z 645.651,A -85,B 0,C 180,E1 7374.032,E2 7374.032} C_VEL
LIN {X 0,Y 370.338,Z 646.293,A -85,B 0,C 180,E1 7373.693,E2 7373.693} C_VEL
LIN {X 0,Y 357.88,Z 751.789,A -85,B 0,C 180,E1 7372.369,E2 7372.369} C_VEL
LIN {X 0,Y 353.035,Z 777.762,A -85,B 0,C 180,E1 7371.985,E2 7371.985} C_VEL
LIN {X 0,Y 347.557,Z 799.413,A -85,B 0,C 180,E1 7371.58,E2 7371.58} C_VEL
LIN {X 0,Y 339.664,Z 824.008,A -85,B 0,C 180,E1 7370.979,E2 7370.979} C_VEL
LIN {X 0,Y 331.666,Z 844.431,A -85,B 0,C 180,E1 7370.34,E2 7370.34} C_VEL
LIN {X 0,Y 321.374,Z 866.861,A -85,B 0,C 180,E1 7369.473,E2 7369.473} C_VEL
LIN {X 0,Y 310.217,Z 887.437,A -85,B 0,C 180,E1 7368.479,E2 7368.479} C_VEL
LIN {X 0,Y 297.782,Z 907.691,A -85,B 0,C 180,E1 7367.275,E2 7367.275} C_VEL
LIN {X 0,Y 284.128,Z 926.943,A -85,B 0,C 180,E1 7365.819,E2 7365.819} C_VEL
LIN {X 0,Y 269.735,Z 945.158,A -85,B 0,C 180,E1 7364.104,E2 7364.104} C_VEL
LIN {X 0,Y 254.375,Z 962.289,A -85,B 0,C 180,E1 7362.035,E2 7362.035} C_VEL
LIN {X 0,Y 239.451,Z 977.364,A -85,B 0,C 180,E1 7359.721,E2 7359.721} C_VEL
LIN {X 0,Y 222.273,Z 992.933,A -85,B 0,C 180,E1 7356.59,E2 7356.59} C_VEL
LIN {X 0,Y 207.108,Z 1005.405,A -85,B 0,C 180,E1 7353.272,E2 7353.272} C_VEL
LIN {X 0,Y 189.492,Z 1018.593,A -85,B 0,C 180,E1 7348.507,E2 7348.507} C_VEL
LIN {X 0,Y 175.853,Z 1027.98,A -85,B 0,C 180,E1 7343.843,E2 7343.843} C_VEL
LIN {X 0,Y 160.888,Z 1037.679,A -85,B 0,C 180,E1 7337.168,E2 7337.168} C_VEL
LIN {X 0,Y 149.223,Z 1044.838,A -85,B 0,C 180,E1 7330.035,E2 7330.035} C_VEL
LIN {X 0,Y 139.232,Z 1051.1,A -85,B 0,C 180,E1 7321.136,E2 7321.136} C_VEL
LIN {X 0,Y 132.661,Z 1055.377,A -85,B 0,C 180,E1 7311.674,E2 7311.674} C_VEL
LIN {X 0,Y 129.421,Z 1057.985,A -85,B 0,C 180,E1 7302.947,E2 7302.947} C_VEL
LIN {X 0,Y 128.164,Z 1059.622,A -85,B 0,C 180,E1 7293.578,E2 7293.578} C_VEL
LIN {X 0,Y 128.058,Z 1060.074,A -85,B 0,C 180,E1 7285.97,E2 7285.97} C_VEL
LIN {X 0,Y 128.626,Z 1059.693,A -85,B 0,C 180,E1 7277.428,E2 7277.428} C_VEL
LIN {X 0,Y 131.235,Z 1057.989,A -85,B 0,C 180,E1 7267.607,E2 7267.607} C_VEL
LIN {X 0,Y 136.337,Z 1055.198,A -85,B 0,C 180,E1 7258.62,E2 7258.62} C_VEL
LIN {X 0,Y 146.26,Z 1050.004,A -85,B 0,C 180,E1 7248.461,E2 7248.461} C_VEL
LIN {X 0,Y 157.505,Z 1044.026,A -85,B 0,C 180,E1 7240.935,E2 7240.935} C_VEL
LIN {X 0,Y 172.914,Z 1035.402,A -85,B 0,C 180,E1 7233.624,E2 7233.624} C_VEL
LIN {X 0,Y 187.59,Z 1026.49,A -85,B 0,C 180,E1 7228.42,E2 7228.42} C_VEL
LIN {X 0,Y 205.337,Z 1014.749,A -85,B 0,C 180,E1 7223.535,E2 7223.535} C_VEL
LIN {X 0,Y 221.332,Z 1003.013,A -85,B 0,C 180,E1 7220.005,E2 7220.005} C_VEL
LIN {X 0,Y 239.151,Z 988.614,A -85,B 0,C 180,E1 7216.768,E2 7216.768} C_VEL
LIN {X 0,Y 254.925,Z 974.31,A -85,B 0,C 180,E1 7214.349,E2 7214.349} C_VEL
LIN {X 0,Y 271.109,Z 958.165,A -85,B 0,C 180,E1 7212.215,E2 7212.215} C_VEL
LIN {X 0,Y 286.688,Z 940.467,A -85,B 0,C 180,E1 7210.411,E2 7210.411} C_VEL
LIN {X 0,Y 301.117,Z 922.247,A -85,B 0,C 180,E1 7208.93,E2 7208.93} C_VEL
LIN {X 0,Y 314.773,Z 902.473,A -85,B 0,C 180,E1 7207.658,E2 7207.658} C_VEL
LIN {X 0,Y 326.215,Z 883.786,A -85,B 0,C 180,E1 7206.689,E2 7206.689} C_VEL
LIN {X 0,Y 338.158,Z 861.218,A -85,B 0,C 180,E1 7205.74,E2 7205.74} C_VEL
LIN {X 0,Y 346.834,Z 842.123,A -85,B 0,C 180,E1 7205.1,E2 7205.1} C_VEL
LIN {X 0,Y 355.55,Z 819.751,A -85,B 0,C 180,E1 7204.485,E2 7204.485} C_VEL
LIN {X 0,Y 362.773,Z 796.484,A -85,B 0,C 180,E1 7203.981,E2 7203.981} C_VEL
LIN {X 0,Y 368.791,Z 772.18,A -85,B 0,C 180,E1 7203.579,E2 7203.579} C_VEL
LIN {X 0,Y 372.984,Z 747.643,A -85,B 0,C 180,E1 7203.258,E2 7203.258} C_VEL
LIN {X 0,Y 383.708,Z 658.313,A -85,B 0,C 180,E1 7202.173,E2 7202.173} C_VEL
LIN {X 0,Y 383.425,Z 656.303,A -85,B 0,C 180,E1 7199.103,E2 7199.103} C_VEL
LIN {X 0,Y 383.701,Z 658.574,A -85,B 0,C 180,E1 7196.091,E2 7196.091} C_VEL
LIN {X 0,Y 372.175,Z 753.84,A -85,B 0,C 180,E1 7194.939,E2 7194.939} C_VEL
LIN {X 0,Y 367.238,Z 779.788,A -85,B 0,C 180,E1 7194.593,E2 7194.593} C_VEL
LIN {X 0,Y 361.55,Z 801.82,A -85,B 0,C 180,E1 7194.266,E2 7194.266} C_VEL
LIN {X 0,Y 353.527,Z 826.276,A -85,B 0,C 180,E1 7193.803,E2 7193.803} C_VEL
LIN {X 0,Y 345.326,Z 846.818,A -85,B 0,C 180,E1 7193.292,E2 7193.292} C_VEL
LIN {X 0,Y 336.89,Z 865.112,A -85,B 0,C 180,E1 7192.734,E2 7192.734} C_VEL
LIN {X 0,Y 333.321,Z 872.022,A -85,B 0,C 180,E1 7192.662,E2 7192.662} C_VEL
LIN {X 0,Y 322.979,Z 889.144,A -85,B 0,C 180,E1 7193.041,E2 7193.041} C_VEL
LIN {X 0,Y 318.967,Z 895.72,A -85,B 0,C 180,E1 7192.933,E2 7192.933} C_VEL
LIN {X 0,Y 305.618,Z 915.782,A -85,B 0,C 180,E1 7191.913,E2 7191.913} C_VEL
LIN {X 0,Y 292.246,Z 933.68,A -85,B 0,C 180,E1 7190.777,E2 7190.777} C_VEL
LIN {X 0,Y 275.862,Z 953.045,A -85,B 0,C 180,E1 7189.194,E2 7189.194} C_VEL
LIN {X 0,Y 261.098,Z 968.605,A -85,B 0,C 180,E1 7187.564,E2 7187.564} C_VEL
LIN {X 0,Y 242.759,Z 985.909,A -85,B 0,C 180,E1 7185.204,E2 7185.204} C_VEL
LIN {X 0,Y 227.108,Z 999.111,A -85,B 0,C 180,E1 7182.821,E2 7182.821} C_VEL
LIN {X 0,Y 209.182,Z 1012.887,A -85,B 0,C 180,E1 7179.534,E2 7179.534} C_VEL
LIN {X 0,Y 192.07,Z 1024.608,A -85,B 0,C 180,E1 7175.648,E2 7175.648} C_VEL
LIN {X 0,Y 175.273,Z 1035.25,A -85,B 0,C 180,E1 7170.789,E2 7170.789} C_VEL
LIN {X 0,Y 159.287,Z 1044.401,A -85,B 0,C 180,E1 7164.691,E2 7164.691} C_VEL
LIN {X 0,Y 145.952,Z 1051.661,A -85,B 0,C 180,E1 7157.722,E2 7157.722} C_VEL
LIN {X 0,Y 133.714,Z 1058.058,A -85,B 0,C 180,E1 7148.365,E2 7148.365} C_VEL
LIN {X 0,Y 126.04,Z 1062.211,A -85,B 0,C 180,E1 7138.942,E2 7138.942} C_VEL
LIN {X 0,Y 121.175,Z 1065.293,A -85,B 0,C 180,E1 7127.281,E2 7127.281} C_VEL
LIN {X 0,Y 120.027,Z 1066.452,A -85,B 0,C 180,E1 7117.66,E2 7117.66} C_VEL
LIN {X 0,Y 120.054,Z 1066.61,A -85,B 0,C 180,E1 7110.477,E2 7110.477} C_VEL
LIN {X 0,Y 120.009,Z 1066.11,A -85,B 0,C 180,E1 7103.302,E2 7103.302} C_VEL
LIN {X 0,Y 120.942,Z 1064.37,A -85,B 0,C 180,E1 7093.675,E2 7093.675} C_VEL
LIN {X 0,Y 124.187,Z 1061.519,A -85,B 0,C 180,E1 7084.229,E2 7084.229} C_VEL
LIN {X 0,Y 131.549,Z 1056.624,A -85,B 0,C 180,E1 7073.639,E2 7073.639} C_VEL
LIN {X 0,Y 141.948,Z 1050.183,A -85,B 0,C 180,E1 7064.647,E2 7064.647} C_VEL
LIN {X 0,Y 155.148,Z 1042.232,A -85,B 0,C 180,E1 7056.951,E2 7056.951} C_VEL
LIN {X 0,Y 170.574,Z 1032.312,A -85,B 0,C 180,E1 7050.492,E2 7050.492} C_VEL
LIN {X 0,Y 187.057,Z 1021.134,A -85,B 0,C 180,E1 7045.317,E2 7045.317} C_VEL
LIN {X 0,Y 203.778,Z 1008.56,A -85,B 0,C 180,E1 7041.207,E2 7041.207} C_VEL
LIN {X 0,Y 219.791,Z 995.518,A -85,B 0,C 180,E1 7038.02,E2 7038.02} C_VEL
LIN {X 0,Y 237.218,Z 979.715,A -85,B 0,C 180,E1 7035.149,E2 7035.149} C_VEL
LIN {X 0,Y 252.175,Z 964.723,A -85,B 0,C 180,E1 7033.062,E2 7033.062} C_VEL
LIN {X 0,Y 269.422,Z 945.358,A -85,B 0,C 180,E1 7030.997,E2 7030.997} C_VEL
LIN {X 0,Y 282.917,Z 928.318,A -85,B 0,C 180,E1 7029.583,E2 7029.583} C_VEL
LIN {X 0,Y 298.008,Z 906.79,A -85,B 0,C 180,E1 7028.191,E2 7028.191} C_VEL
LIN {X 0,Y 309.442,Z 888.158,A -85,B 0,C 180,E1 7027.24,E2 7027.24} C_VEL
LIN {X 0,Y 320.947,Z 866.883,A -85,B 0,C 180,E1 7026.371,E2 7026.371} C_VEL
LIN {X 0,Y 330.595,Z 845.825,A -85,B 0,C 180,E1 7025.694,E2 7025.694} C_VEL
LIN {X 0,Y 339.323,Z 823.637,A -85,B 0,C 180,E1 7025.132,E2 7025.132} C_VEL
LIN {X 0,Y 346.957,Z 799.492,A -85,B 0,C 180,E1 7024.671,E2 7024.671} C_VEL
LIN {X 0,Y 352.661,Z 776.787,A -85,B 0,C 180,E1 7024.327,E2 7024.327} C_VEL
LIN {X 0,Y 357.229,Z 751.21,A -85,B 0,C 180,E1 7023.983,E2 7023.983} C_VEL
LIN {X 0,Y 368.955,Z 652.825,A -85,B 0,C 180,E1 7022.757,E2 7022.757} C_VEL
LIN {X 0,Y 368.401,Z 650.188,A -85,B 0,C 180,E1 7018.6,E2 7018.6} C_VEL
LIN {X 0,Y 368.922,Z 652.997,A -85,B 0,C 180,E1 7014.851,E2 7014.851} C_VEL
LIN {X 0,Y 357.03,Z 752.129,A -85,B 0,C 180,E1 7013.644,E2 7013.644} C_VEL
LIN {X 0,Y 352.162,Z 777.923,A -85,B 0,C 180,E1 7013.279,E2 7013.279} C_VEL
LIN {X 0,Y 346.624,Z 799.601,A -85,B 0,C 180,E1 7012.894,E2 7012.894} C_VEL
LIN {X 0,Y 338.504,Z 824.588,A -85,B 0,C 180,E1 7012.313,E2 7012.313} C_VEL
LIN {X 0,Y 330.419,Z 844.968,A -85,B 0,C 180,E1 7011.706,E2 7011.706} C_VEL
LIN {X 0,Y 320.007,Z 867.333,A -85,B 0,C 180,E1 7010.883,E2 7010.883} C_VEL
LIN {X 0,Y 309.183,Z 887.081,A -85,B 0,C 180,E1 7009.979,E2 7009.979} C_VEL
LIN {X 0,Y 296.578,Z 907.398,A -85,B 0,C 180,E1 7008.837,E2 7008.837} C_VEL
LIN {X 0,Y 282.72,Z 926.733,A -85,B 0,C 180,E1 7007.454,E2 7007.454} C_VEL
LIN {X 0,Y 268.801,Z 944.121,A -85,B 0,C 180,E1 7005.906,E2 7005.906} C_VEL
LIN {X 0,Y 252.885,Z 961.726,A -85,B 0,C 180,E1 7003.905,E2 7003.905} C_VEL
LIN {X 0,Y 237.947,Z 976.565,A -85,B 0,C 180,E1 7001.748,E2 7001.748} C_VEL
LIN {X 0,Y 219.788,Z 992.744,A -85,B 0,C 180,E1 6998.657,E2 6998.657} C_VEL
LIN {X 0,Y 204.377,Z 1005.091,A -85,B 0,C 180,E1 6995.502,E2 6995.502} C_VEL
LIN {X 0,Y 186.421,Z 1018.179,A -85,B 0,C 180,E1 6990.958,E2 6990.958} C_VEL
LIN {X 0,Y 171.165,Z 1028.266,A -85,B 0,C 180,E1 6986.049,E2 6986.049} C_VEL
LIN {X 0,Y 155.456,Z 1037.949,A -85,B 0,C 180,E1 6979.374,E2 6979.374} C_VEL
LIN {X 0,Y 143.079,Z 1045.101,A -85,B 0,C 180,E1 6972.135,E2 6972.135} C_VEL
LIN {X 0,Y 132.341,Z 1051.348,A -85,B 0,C 180,E1 6962.955,E2 6962.955} C_VEL
LIN {X 0,Y 125.175,Z 1055.616,A -85,B 0,C 180,E1 6953.042,E2 6953.042} C_VEL
LIN {X 0,Y 121.589,Z 1058.217,A -85,B 0,C 180,E1 6943.797,E2 6943.797} C_VEL
LIN {X 0,Y 120.176,Z 1059.846,A -85,B 0,C 180,E1 6933.816,E2 6933.816} C_VEL
LIN {X 0,Y 120.057,Z 1060.267,A -85,B 0,C 180,E1 6926.18,E2 6926.18} C_VEL
LIN {X 0,Y 120.6,Z 1059.997,A -85,B 0,C 180,E1 6917.551,E2 6917.551} C_VEL
LIN {X 0,Y 123.513,Z 1058.299,A -85,B 0,C 180,E1 6906.629,E2 6906.629} C_VEL
LIN {X 0,Y 129.043,Z 1055.548,A -85,B 0,C 180,E1 6897.153,E2 6897.153} C_VEL
LIN {X 0,Y 139.206,Z 1050.684,A -85,B 0,C 180,E1 6886.971,E2 6886.971} C_VEL
LIN {X 0,Y 151.012,Z 1044.796,A -85,B 0,C 180,E1 6879.223,E2 6879.223} C_VEL
LIN {X 0,Y 166.39,Z 1036.761,A -85,B 0,C 180,E1 6872.079,E2 6872.079} C_VEL
LIN {X 0,Y 182.271,Z 1027.55,A -85,B 0,C 180,E1 6866.597,E2 6866.597} C_VEL
LIN {X 0,Y 199.512,Z 1016.739,A -85,B 0,C 180,E1 6862.004,E2 6862.004} C_VEL
LIN {X 0,Y 217.197,Z 1004.209,A -85,B 0,C 180,E1 6858.243,E2 6858.243} C_VEL
LIN {X 0,Y 235.133,Z 990.253,A -85,B 0,C 180,E1 6855.137,E2 6855.137} C_VEL
LIN {X 0,Y 252.107,Z 975.246,A -85,B 0,C 180,E1 6852.665,E2 6852.665} C_VEL
LIN {X 0,Y 267.644,Z 960.101,A -85,B 0,C 180,E1 6850.723,E2 6850.723} C_VEL
LIN {X 0,Y 283.449,Z 942.74,A -85,B 0,C 180,E1 6848.987,E2 6848.987} C_VEL
LIN {X 0,Y 296.637,Z 926.541,A -85,B 0,C 180,E1 6847.693,E2 6847.693} C_VEL
LIN {X 0,Y 311.398,Z 906.15,A -85,B 0,C 180,E1 6846.386,E2 6846.386} C_VEL
LIN {X 0,Y 323.41,Z 887.065,A -85,B 0,C 180,E1 6845.419,E2 6845.419} C_VEL
LIN {X 0,Y 335.02,Z 866.15,A -85,B 0,C 180,E1 6844.552,E2 6844.552} C_VEL
LIN {X 0,Y 345.476,Z 843.715,A -85,B 0,C 180,E1 6843.817,E2 6843.817} C_VEL
LIN {X 0,Y 354.205,Z 821.776,A -85,B 0,C 180,E1 6843.237,E2 6843.237} C_VEL
LIN {X 0,Y 361.842,Z 797.83,A -85,B 0,C 180,E1 6842.739,E2 6842.739} C_VEL
LIN {X 0,Y 367.588,Z 775.195,A -85,B 0,C 180,E1 6842.377,E2 6842.377} C_VEL
LIN {X 0,Y 372.198,Z 749.776,A -85,B 0,C 180,E1 6842.054,E2 6842.054} C_VEL
LIN {X 0,Y 382.496,Z 665.556,A -85,B 0,C 180,E1 6841.049,E2 6841.049} C_VEL
LIN {X 0,Y 382.444,Z 664.293,A -85,B 0,C 180,E1 6839.101,E2 6839.101} C_VEL
LIN {X 0,Y 382.492,Z 665.732,A -85,B 0,C 180,E1 6837.205,E2 6837.205} C_VEL
LIN {X 0,Y 371.661,Z 753.865,A -85,B 0,C 180,E1 6836.171,E2 6836.171} C_VEL
LIN {X 0,Y 366.66,Z 779.786,A -85,B 0,C 180,E1 6835.842,E2 6835.842} C_VEL
LIN {X 0,Y 360.9,Z 801.879,A -85,B 0,C 180,E1 6835.534,E2 6835.534} C_VEL
LIN {X 0,Y 352.752,Z 826.425,A -85,B 0,C 180,E1 6835.098,E2 6835.098} C_VEL
LIN {X 0,Y 344.162,Z 847.662,A -85,B 0,C 180,E1 6834.6,E2 6834.6} C_VEL
LIN {X 0,Y 332.852,Z 871.234,A -85,B 0,C 180,E1 6833.894,E2 6833.894} C_VEL
LIN {X 0,Y 322.247,Z 890.168,A -85,B 0,C 180,E1 6833.177,E2 6833.177} C_VEL
LIN {X 0,Y 318.967,Z 895.72,A -85,B 0,C 180,E1 6832.933,E2 6832.933} C_VEL
LIN {X 0,Y 314.839,Z 902.268,A -85,B 0,C 180,E1 6832.811,E2 6832.811} C_VEL
LIN {X 0,Y 302.976,Z 918.459,A -85,B 0,C 180,E1 6833.094,E2 6833.094} C_VEL
LIN {X 0,Y 298.215,Z 924.523,A -85,B 0,C 180,E1 6832.932,E2 6832.932} C_VEL
LIN {X 0,Y 283.914,Z 942.227,A -85,B 0,C 180,E1 6831.74,E2 6831.74} C_VEL
LIN {X 0,Y 268.808,Z 959.07,A -85,B 0,C 180,E1 6830.308,E2 6830.308} C_VEL
LIN {X 0,Y 251.122,Z 976.489,A -85,B 0,C 180,E1 6828.378,E2 6828.378} C_VEL
LIN {X 0,Y 235.585,Z 990.243,A -85,B 0,C 180,E1 6826.395,E2 6826.395} C_VEL
LIN {X 0,Y 215.985,Z 1005.771,A -85,B 0,C 180,E1 6823.395,E2 6823.395} C_VEL
LIN {X 0,Y 199.626,Z 1017.375,A -85,B 0,C 180,E1 6820.332,E2 6820.332} C_VEL
LIN {X 0,Y 180.741,Z 1029.519,A -85,B 0,C 180,E1 6815.897,E2 6815.897} C_VEL
LIN {X 0,Y 164.156,Z 1039.091,A -85,B 0,C 180,E1 6810.837,E2 6810.837} C_VEL
LIN {X 0,Y 147.965,Z 1047.771,A -85,B 0,C 180,E1 6804.185,E2 6804.185} C_VEL
LIN {X 0,Y 134.062,Z 1054.604,A -85,B 0,C 180,E1 6796.081,E2 6796.081} C_VEL
LIN {X 0,Y 122.722,Z 1060.188,A -85,B 0,C 180,E1 6785.918,E2 6785.918} C_VEL
LIN {X 0,Y 115.501,Z 1063.804,A -85,B 0,C 180,E1 6774.553,E2 6774.553} C_VEL
LIN {X 0,Y 112.579,Z 1065.671,A -85,B 0,C 180,E1 6764.4,E2 6764.4} C_VEL
LIN {X 0,Y 112.006,Z 1066.421,A -85,B 0,C 180,E1 6754.608,E2 6754.608} C_VEL
LIN {X 0,Y 112.038,Z 1066.28,A -85,B 0,C 180,E1 6747.954,E2 6747.954} C_VEL
LIN {X 0,Y 112.075,Z 1065.601,A -85,B 0,C 180,E1 6740.759,E2 6740.759} C_VEL
LIN {X 0,Y 113.391,Z 1063.899,A -85,B 0,C 180,E1 6731.491,E2 6731.491} C_VEL
LIN {X 0,Y 117.932,Z 1060.613,A -85,B 0,C 180,E1 6720.544,E2 6720.544} C_VEL
LIN {X 0,Y 126.723,Z 1055.319,A -85,B 0,C 180,E1 6709.683,E2 6709.683} C_VEL
LIN {X 0,Y 137.945,Z 1048.984,A -85,B 0,C 180,E1 6701.076,E2 6701.076} C_VEL
LIN {X 0,Y 153.657,Z 1039.893,A -85,B 0,C 180,E1 6692.919,E2 6692.919} C_VEL
LIN {X 0,Y 168.008,Z 1031.088,A -85,B 0,C 180,E1 6687.531,E2 6687.531} C_VEL
LIN {X 0,Y 185.99,Z 1019.157,A -85,B 0,C 180,E1 6682.38,E2 6682.38} C_VEL
LIN {X 0,Y 202.629,Z 1006.956,A -85,B 0,C 180,E1 6678.659,E2 6678.659} C_VEL
LIN {X 0,Y 220.875,Z 992.242,A -85,B 0,C 180,E1 6675.369,E2 6675.369} C_VEL
LIN {X 0,Y 237.01,Z 977.66,A -85,B 0,C 180,E1 6672.959,E2 6672.959} C_VEL
LIN {X 0,Y 253.983,Z 960.747,A -85,B 0,C 180,E1 6670.814,E2 6670.814} C_VEL
LIN {X 0,Y 269.384,Z 943.299,A -85,B 0,C 180,E1 6669.131,E2 6669.131} C_VEL
LIN {X 0,Y 284.049,Z 924.85,A -85,B 0,C 180,E1 6667.729,E2 6667.729} C_VEL
LIN {X 0,Y 297.961,Z 904.806,A -85,B 0,C 180,E1 6666.552,E2 6666.552} C_VEL
LIN {X 0,Y 309.928,Z 885.325,A -85,B 0,C 180,E1 6665.635,E2 6665.635} C_VEL
LIN {X 0,Y 322.091,Z 862.325,A -85,B 0,C 180,E1 6664.793,E2 6664.793} C_VEL
LIN {X 0,Y 330.868,Z 843.009,A -85,B 0,C 180,E1 6664.238,E2 6664.238} C_VEL
LIN {X 0,Y 340.118,Z 818.907,A -85,B 0,C 180,E1 6663.69,E2 6663.69} C_VEL
LIN {X 0,Y 346.949,Z 796.809,A -85,B 0,C 180,E1 6663.31,E2 6663.31} C_VEL
LIN {X 0,Y 352.996,Z 771.961,A -85,B 0,C 180,E1 6662.964,E2 6662.964} C_VEL
LIN {X 0,Y 356.987,Z 748.391,A -85,B 0,C 180,E1 6662.666,E2 6662.666} C_VEL
LIN {X 0,Y 367.625,Z 660.061,A -85,B 0,C 180,E1 6661.598,E2 6661.598} C_VEL
LIN {X 0,Y 367.418,Z 658.194,A -85,B 0,C 180,E1 6658.597,E2 6658.597} C_VEL
LIN {X 0,Y 367.593,Z 660.258,A -85,B 0,C 180,E1 6656.011,E2 6656.011} C_VEL
LIN {X 0,Y 356.344,Z 752.576,A -85,B 0,C 180,E1 6654.922,E2 6654.922} C_VEL
LIN {X 0,Y 351.41,Z 778.343,A -85,B 0,C 180,E1 6654.575,E2 6654.575} C_VEL
LIN {X 0,Y 345.789,Z 800.094,A -85,B 0,C 180,E1 6654.209,E2 6654.209} C_VEL
LIN {X 0,Y 337.529,Z 825.168,A -85,B 0,C 180,E1 6653.656,E2 6653.656} C_VEL
LIN {X 0,Y 329.361,Z 845.504,A -85,B 0,C 180,E1 6653.082,E2 6653.082} C_VEL
LIN {X 0,Y 318.359,Z 868.696,A -85,B 0,C 180,E1 6652.269,E2 6652.269} C_VEL
LIN {X 0,Y 307.414,Z 888.331,A -85,B 0,C 180,E1 6651.41,E2 6651.41} C_VEL
LIN {X 0,Y 294.186,Z 909.18,A -85,B 0,C 180,E1 6650.285,E2 6650.285} C_VEL
LIN {X 0,Y 280.149,Z 928.327,A -85,B 0,C 180,E1 6648.965,E2 6648.965} C_VEL
LIN {X 0,Y 264.823,Z 946.994,A -85,B 0,C 180,E1 6647.35,E2 6647.35} C_VEL
LIN {X 0,Y 248.953,Z 963.905,A -85,B 0,C 180,E1 6645.454,E2 6645.454} C_VEL
LIN {X 0,Y 231.999,Z 980.229,A -85,B 0,C 180,E1 6643.096,E2 6643.096} C_VEL
LIN {X 0,Y 214.615,Z 994.953,A -85,B 0,C 180,E1 6640.24,E2 6640.24} C_VEL
LIN {X 0,Y 197.025,Z 1008.519,A -85,B 0,C 180,E1 6636.717,E2 6636.717} C_VEL
LIN {X 0,Y 179.49,Z 1020.493,A -85,B 0,C 180,E1 6632.343,E2 6632.343} C_VEL
LIN {X 0,Y 163.159,Z 1030.799,A -85,B 0,C 180,E1 6627.095,E2 6627.095} C_VEL
LIN {X 0,Y 147.671,Z 1039.631,A -85,B 0,C 180,E1 6620.47,E2 6620.47} C_VEL
LIN {X 0,Y 135.006,Z 1046.546,A -85,B 0,C 180,E1 6612.951,E2 6612.951} C_VEL
LIN {X 0,Y 123.605,Z 1052.596,A -85,B 0,C 180,E1 6602.819,E2 6602.819} C_VEL
LIN {X 0,Y 117.004,Z 1056.319,A -85,B 0,C 180,E1 6593.148,E2 6593.148} C_VEL
LIN {X 0,Y 113.087,Z 1059.089,A -85,B 0,C 180,E1 6581.733,E2 6581.733} C_VEL
LIN {X 0,Y 112.1,Z 1060.233,A -85,B 0,C 180,E1 6571.533,E2 6571.533} C_VEL
LIN {X 0,Y 112.139,Z 1060.466,A -85,B 0,C 180,E1 6563.344,E2 6563.344} C_VEL
LIN {X 0,Y 113.251,Z 1059.849,A -85,B 0,C 180,E1 6553.589,E2 6553.589} C_VEL
LIN {X 0,Y 116.739,Z 1058.174,A -85,B 0,C 180,E1 6543.552,E2 6543.552} C_VEL
LIN {X 0,Y 124.512,Z 1054.812,A -85,B 0,C 180,E1 6532.388,E2 6532.388} C_VEL
LIN {X 0,Y 135.935,Z 1049.623,A -85,B 0,C 180,E1 6522.645,E2 6522.645} C_VEL
LIN {X 0,Y 150.415,Z 1042.886,A -85,B 0,C 180,E1 6514.483,E2 6514.483} C_VEL
LIN {X 0,Y 166.507,Z 1034.524,A -85,B 0,C 180,E1 6508.024,E2 6508.024} C_VEL
LIN {X 0,Y 183.473,Z 1024.981,A -85,B 0,C 180,E1 6502.925,E2 6502.925} C_VEL
LIN {X 0,Y 201.597,Z 1013.472,A -85,B 0,C 180,E1 6498.678,E2 6498.678} C_VEL
LIN {X 0,Y 217.988,Z 1002.004,A -85,B 0,C 180,E1 6495.581,E2 6495.581} C_VEL
LIN {X 0,Y 236.723,Z 987.299,A -85,B 0,C 180,E1 6492.652,E2 6492.652} C_VEL
LIN {X 0,Y 252.276,Z 973.658,A -85,B 0,C 180,E1 6490.598,E2 6490.598} C_VEL
LIN {X 0,Y 269.993,Z 956.293,A -85,B 0,C 180,E1 6488.581,E2 6488.581} C_VEL
LIN {X 0,Y 284.664,Z 940.026,A -85,B 0,C 180,E1 6487.12,E2 6487.12} C_VEL
LIN {X 0,Y 299.5,Z 921.709,A -85,B 0,C 180,E1 6485.8,E2 6485.8} C_VEL
LIN {X 0,Y 313.488,Z 901.774,A -85,B 0,C 180,E1 6484.672,E2 6484.672} C_VEL
LIN {X 0,Y 326.161,Z 881.362,A -85,B 0,C 180,E1 6483.745,E2 6483.745} C_VEL
LIN {X 0,Y 337.414,Z 860.061,A -85,B 0,C 180,E1 6482.964,E2 6482.964} C_VEL
LIN {X 0,Y 346.758,Z 839.635,A -85,B 0,C 180,E1 6482.367,E2 6482.367} C_VEL
LIN {X 0,Y 355.888,Z 815.615,A -85,B 0,C 180,E1 6481.808,E2 6481.808} C_VEL
LIN {X 0,Y 362.296,Z 794.911,A -85,B 0,C 180,E1 6481.42,E2 6481.42} C_VEL
LIN {X 0,Y 368.455,Z 769.444,A -85,B 0,C 180,E1 6481.052,E2 6481.052} C_VEL
LIN {X 0,Y 372.322,Z 746.73,A -85,B 0,C 180,E1 6480.784,E2 6480.784} C_VEL
LIN {X 0,Y 381.439,Z 672.756,A -85,B 0,C 180,E1 6479.932,E2 6479.932} C_VEL
LIN {X 0,Y 381.452,Z 672.386,A -85,B 0,C 180,E1 6478.949,E2 6478.949} C_VEL
LIN {X 0,Y 381.42,Z 672.966,A -85,B 0,C 180,E1 6478.325,E2 6478.325} C_VEL
LIN {X 0,Y 371.322,Z 753.862,A -85,B 0,C 180,E1 6477.407,E2 6477.407} C_VEL
LIN {X 0,Y 366.297,Z 779.61,A -85,B 0,C 180,E1 6477.097,E2 6477.097} C_VEL
LIN {X 0,Y 360.488,Z 801.723,A -85,B 0,C 180,E1 6476.808,E2 6476.808} C_VEL
LIN {X 0,Y 352.157,Z 826.574,A -85,B 0,C 180,E1 6476.398,E2 6476.398} C_VEL
LIN {X 0,Y 343.82,Z 847.028,A -85,B 0,C 180,E1 6475.951,E2 6475.951} C_VEL
LIN {X 0,Y 332.579,Z 870.374,A -85,B 0,C 180,E1 6475.305,E2 6475.305} C_VEL
LIN {X 0,Y 321.873,Z 889.371,A -85,B 0,C 180,E1 6474.639,E2 6474.639} C_VEL
LIN {X 0,Y 308.812,Z 909.865,A -85,B 0,C 180,E1 6473.733,E2 6473.733} C_VEL
LIN {X 0,Y 298.215,Z 924.523,A -85,B 0,C 180,E1 6472.932,E2 6472.932} C_VEL
LIN {X 0,Y 293.351,Z 930.543,A -85,B 0,C 180,E1 6472.753,E2 6472.753} C_VEL
LIN {X 0,Y 280.073,Z 945.633,A -85,B 0,C 180,E1 6472.924,E2 6472.924} C_VEL
LIN {X 0,Y 274.85,Z 951.223,A -85,B 0,C 180,E1 6472.694,E2 6472.694} C_VEL
LIN {X 0,Y 259.962,Z 966.576,A -85,B 0,C 180,E1 6471.301,E2 6471.301} C_VEL
LIN {X 0,Y 243.062,Z 982.334,A -85,B 0,C 180,E1 6469.477,E2 6469.477} C_VEL
LIN {X 0,Y 224.624,Z 997.462,A -85,B 0,C 180,E1 6467.125,E2 6467.125} C_VEL
LIN {X 0,Y 207.534,Z 1010.121,A -85,B 0,C 180,E1 6464.491,E2 6464.491} C_VEL
LIN {X 0,Y 187.816,Z 1023.112,A -85,B 0,C 180,E1 6460.727,E2 6460.727} C_VEL
LIN {X 0,Y 171.005,Z 1033.081,A -85,B 0,C 180,E1 6456.636,E2 6456.636} C_VEL
LIN {X 0,Y 151.605,Z 1043.422,A -85,B 0,C 180,E1 6450.353,E2 6450.353} C_VEL
LIN {X 0,Y 136.803,Z 1050.604,A -85,B 0,C 180,E1 6443.699,E2 6443.699} C_VEL
LIN {X 0,Y 121.687,Z 1057.462,A -85,B 0,C 180,E1 6433.648,E2 6433.648} C_VEL
LIN {X 0,Y 112.63,Z 1061.485,A -85,B 0,C 180,E1 6424.007,E2 6424.007} C_VEL
LIN {X 0,Y 106.212,Z 1064.656,A -85,B 0,C 180,E1 6411.54,E2 6411.54} C_VEL
LIN {X 0,Y 104.081,Z 1066.001,A -85,B 0,C 180,E1 6399.399,E2 6399.399} C_VEL
LIN {X 0,Y 104.052,Z 1066.199,A -85,B 0,C 180,E1 6391.101,E2 6391.101} C_VEL
LIN {X 0,Y 104.011,Z 1065.803,A -85,B 0,C 180,E1 6383.376,E2 6383.376} C_VEL
LIN {X 0,Y 105.268,Z 1064.022,A -85,B 0,C 180,E1 6371.733,E2 6371.733} C_VEL
LIN {X 0,Y 109.344,Z 1061.202,A -85,B 0,C 180,E1 6361.01,E2 6361.01} C_VEL
LIN {X 0,Y 118.19,Z 1056.373,A -85,B 0,C 180,E1 6349.351,E2 6349.351} C_VEL
LIN {X 0,Y 130.239,Z 1049.966,A -85,B 0,C 180,E1 6339.849,E2 6339.849} C_VEL
LIN {X 0,Y 145.069,Z 1042.054,A -85,B 0,C 180,E1 6332.029,E2 6332.029} C_VEL
LIN {X 0,Y 162,Z 1032.205,A -85,B 0,C 180,E1 6325.692,E2 6325.692} C_VEL
LIN {X 0,Y 178.876,Z 1021.623,A -85,B 0,C 180,E1 6320.962,E2 6320.962} C_VEL
LIN {X 0,Y 197.515,Z 1008.582,A -85,B 0,C 180,E1 6316.906,E2 6316.906} C_VEL
LIN {X 0,Y 214.32,Z 995.612,A -85,B 0,C 180,E1 6313.975,E2 6313.975} C_VEL
LIN {X 0,Y 232.528,Z 979.889,A -85,B 0,C 180,E1 6311.358,E2 6311.358} C_VEL
LIN {X 0,Y 247.507,Z 965.482,A -85,B 0,C 180,E1 6309.534,E2 6309.534} C_VEL
LIN {X 0,Y 264.395,Z 947.414,A -85,B 0,C 180,E1 6307.765,E2 6307.765} C_VEL
LIN {X 0,Y 279.214,Z 929.377,A -85,B 0,C 180,E1 6306.408,E2 6306.408} C_VEL
LIN {X 0,Y 293.651,Z 909.717,A -85,B 0,C 180,E1 6305.254,E2 6305.254} C_VEL
LIN {X 0,Y 306.829,Z 888.911,A -85,B 0,C 180,E1 6304.298,E2 6304.298} C_VEL
LIN {X 0,Y 318.904,Z 867.215,A -85,B 0,C 180,E1 6303.517,E2 6303.517} C_VEL
LIN {X 0,Y 328.89,Z 845.887,A -85,B 0,C 180,E1 6302.919,E2 6302.919} C_VEL
LIN {X 0,Y 337.766,Z 823.768,A -85,B 0,C 180,E1 6302.43,E2 6302.43} C_VEL
LIN {X 0,Y 345.646,Z 799.384,A -85,B 0,C 180,E1 6302.025,E2 6302.025} C_VEL
LIN {X 0,Y 351.371,Z 777.037,A -85,B 0,C 180,E1 6301.729,E2 6301.729} C_VEL
LIN {X 0,Y 356.147,Z 751.089,A -85,B 0,C 180,E1 6301.412,E2 6301.412} C_VEL
LIN {X 0,Y 366.455,Z 667.232,A -85,B 0,C 180,E1 6300.43,E2 6300.43} C_VEL
LIN {X 0,Y 366.435,Z 666.197,A -85,B 0,C 180,E1 6298.593,E2 6298.593} C_VEL
LIN {X 0,Y 366.428,Z 667.409,A -85,B 0,C 180,E1 6297.18,E2 6297.18} C_VEL
LIN {X 0,Y 355.835,Z 753.023,A -85,B 0,C 180,E1 6296.204,E2 6296.204} C_VEL
LIN {X 0,Y 350.869,Z 778.634,A -85,B 0,C 180,E1 6295.877,E2 6295.877} C_VEL
LIN {X 0,Y 345.198,Z 800.372,A -85,B 0,C 180,E1 6295.533,E2 6295.533} C_VEL
LIN {X 0,Y 336.741,Z 825.748,A -85,B 0,C 180,E1 6295.006,E2 6295.006} C_VEL
LIN {X 0,Y 328.495,Z 846.041,A -85,B 0,C 180,E1 6294.466,E2 6294.466} C_VEL
LIN {X 0,Y 317.38,Z 869.168,A -85,B 0,C 180,E1 6293.702,E2 6293.702} C_VEL
LIN {X 0,Y 306.319,Z 888.777,A -85,B 0,C 180,E1 6292.895,E2 6292.895} C_VEL
LIN {X 0,Y 292.936,Z 909.586,A -85,B 0,C 180,E1 6291.836,E2 6291.836} C_VEL
LIN {X 0,Y 279.066,Z 928.274,A -85,B 0,C 180,E1 6290.623,E2 6290.623} C_VEL
LIN {X 0,Y 263.71,Z 946.77,A -85,B 0,C 180,E1 6289.121,E2 6289.121} C_VEL
LIN {X 0,Y 247.964,Z 963.341,A -85,B 0,C 180,E1 6287.379,E2 6287.379} C_VEL
LIN {X 0,Y 232.474,Z 978.078,A -85,B 0,C 180,E1 6285.407,E2 6285.407} C_VEL
LIN {X 0,Y 213.759,Z 993.892,A -85,B 0,C 180,E1 6282.6,E2 6282.6} C_VEL
LIN {X 0,Y 197.329,Z 1006.337,A -85,B 0,C 180,E1 6279.622,E2 6279.622} C_VEL
LIN {X 0,Y 178.265,Z 1019.27,A -85,B 0,C 180,E1 6275.321,E2 6275.321} C_VEL
LIN {X 0,Y 162.616,Z 1028.836,A -85,B 0,C 180,E1 6270.824,E2 6270.824} C_VEL
LIN {X 0,Y 145.087,Z 1038.627,A -85,B 0,C 180,E1 6264.141,E2 6264.141} C_VEL
LIN {X 0,Y 131.446,Z 1045.626,A -85,B 0,C 180,E1 6256.908,E2 6256.908} C_VEL
LIN {X 0,Y 119.026,Z 1051.843,A -85,B 0,C 180,E1 6247.217,E2 6247.217} C_VEL
LIN {X 0,Y 110.456,Z 1056.096,A -85,B 0,C 180,E1 6236.332,E2 6236.332} C_VEL
LIN {X 0,Y 106.007,Z 1058.689,A -85,B 0,C 180,E1 6225.824,E2 6225.824} C_VEL
LIN {X 0,Y 104.206,Z 1060.293,A -85,B 0,C 180,E1 6214.402,E2 6214.402} C_VEL
LIN {X 0,Y 104.07,Z 1060.702,A -85,B 0,C 180,E1 6205.592,E2 6205.592} C_VEL
LIN {X 0,Y 104.839,Z 1060.422,A -85,B 0,C 180,E1 6195.642,E2 6195.642} C_VEL
LIN {X 0,Y 108.699,Z 1058.693,A -85,B 0,C 180,E1 6183.161,E2 6183.161} C_VEL
LIN {X 0,Y 115.543,Z 1055.941,A -85,B 0,C 180,E1 6172.716,E2 6172.716} C_VEL
LIN {X 0,Y 128.07,Z 1050.846,A -85,B 0,C 180,E1 6161.577,E2 6161.577} C_VEL
LIN {X 0,Y 141.11,Z 1045.148,A -85,B 0,C 180,E1 6153.999,E2 6153.999} C_VEL
LIN {X 0,Y 157.66,Z 1037.371,A -85,B 0,C 180,E1 6147.17,E2 6147.17} C_VEL
LIN {X 0,Y 174.66,Z 1028.309,A -85,B 0,C 180,E1 6141.965,E2 6141.965} C_VEL
LIN {X 0,Y 192.199,Z 1018.053,A -85,B 0,C 180,E1 6137.818,E2 6137.818} C_VEL
LIN {X 0,Y 211.107,Z 1005.519,A -85,B 0,C 180,E1 6134.258,E2 6134.258} C_VEL
LIN {X 0,Y 227.706,Z 993.281,A -85,B 0,C 180,E1 6131.699,E2 6131.699} C_VEL
LIN {X 0,Y 247.145,Z 977.121,A -85,B 0,C 180,E1 6129.189,E2 6129.189} C_VEL
LIN {X 0,Y 263.18,Z 962.114,A -85,B 0,C 180,E1 6127.429,E2 6127.429} C_VEL
LIN {X 0,Y 281.13,Z 943.115,A -85,B 0,C 180,E1 6125.715,E2 6125.715} C_VEL
LIN {X 0,Y 294.897,Z 926.623,A -85,B 0,C 180,E1 6124.549,E2 6124.549} C_VEL
LIN {X 0,Y 310.01,Z 906.158,A -85,B 0,C 180,E1 6123.396,E2 6123.396} C_VEL
LIN {X 0,Y 322.282,Z 887.027,A -85,B 0,C 180,E1 6122.544,E2 6122.544} C_VEL
LIN {X 0,Y 334.124,Z 866.025,A -85,B 0,C 180,E1 6121.779,E2 6121.779} C_VEL
LIN {X 0,Y 344.531,Z 844.055,A -85,B 0,C 180,E1 6121.149,E2 6121.149} C_VEL
LIN {X 0,Y 353.231,Z 822.577,A -85,B 0,C 180,E1 6120.649,E2 6120.649} C_VEL
LIN {X 0,Y 361.031,Z 798.65,A -85,B 0,C 180,E1 6120.207,E2 6120.207} C_VEL
LIN {X 0,Y 366.804,Z 776.382,A -85,B 0,C 180,E1 6119.891,E2 6119.891} C_VEL
LIN {X 0,Y 371.625,Z 750.591,A -85,B 0,C 180,E1 6119.593,E2 6119.593} C_VEL
LIN {X 0,Y 376.911,Z 709.347,A -85,B 0,C 180,E1 6119.134,E2 6119.134} C_VEL
LIN {X 0,Y 370.706,Z 756.915,A -85,B 0,C 180,E1 6118.61,E2 6118.61} C_VEL
LIN {X 0,Y 365.621,Z 781.488,A -85,B 0,C 180,E1 6118.329,E2 6118.329} C_VEL
LIN {X 0,Y 359.172,Z 805.343,A -85,B 0,C 180,E1 6118.034,E2 6118.034} C_VEL
LIN {X 0,Y 351.25,Z 828.005,A -85,B 0,C 180,E1 6117.678,E2 6117.678} C_VEL
LIN {X 0,Y 342.853,Z 848.262,A -85,B 0,C 180,E1 6117.264,E2 6117.264} C_VEL
LIN {X 0,Y 331.525,Z 871.314,A -85,B 0,C 180,E1 6116.664,E2 6116.664} C_VEL
LIN {X 0,Y 320.729,Z 890.198,A -85,B 0,C 180,E1 6116.043,E2 6116.043} C_VEL
LIN {X 0,Y 307.059,Z 911.202,A -85,B 0,C 180,E1 6115.166,E2 6115.166} C_VEL
LIN {X 0,Y 292.984,Z 929.939,A -85,B 0,C 180,E1 6114.169,E2 6114.169} C_VEL
LIN {X 0,Y 277.582,Z 948.286,A -85,B 0,C 180,E1 6112.927,E2 6112.927} C_VEL
LIN {X 0,Y 274.85,Z 951.223,A -85,B 0,C 180,E1 6112.694,E2 6112.694} C_VEL
LIN {X 0,Y 269.489,Z 956.787,A -85,B 0,C 180,E1 6112.442,E2 6112.442} C_VEL
LIN {X 0,Y 253.992,Z 971.308,A -85,B 0,C 180,E1 6112.458,E2 6112.458} C_VEL
LIN {X 0,Y 249.133,Z 975.585,A -85,B 0,C 180,E1 6112.165,E2 6112.165} C_VEL
LIN {X 0,Y 232.222,Z 990.065,A -85,B 0,C 180,E1 6110.333,E2 6110.333} C_VEL
LIN {X 0,Y 211.862,Z 1005.514,A -85,B 0,C 180,E1 6107.673,E2 6107.673} C_VEL
LIN {X 0,Y 194.686,Z 1017.099,A -85,B 0,C 180,E1 6104.917,E2 6104.917} C_VEL
LIN {X 0,Y 174.635,Z 1029.209,A -85,B 0,C 180,E1 6100.861,E2 6100.861} C_VEL
LIN {X 0,Y 157.259,Z 1038.502,A -85,B 0,C 180,E1 6096.289,E2 6096.289} C_VEL
LIN {X 0,Y 138.955,Z 1047.398,A -85,B 0,C 180,E1 6089.755,E2 6089.755} C_VEL
LIN {X 0,Y 123.418,Z 1054.125,A -85,B 0,C 180,E1 6081.8,E2 6081.8} C_VEL
LIN {X 0,Y 110.255,Z 1059.612,A -85,B 0,C 180,E1 6071.455,E2 6071.455} C_VEL
LIN {X 0,Y 101.103,Z 1063.279,A -85,B 0,C 180,E1 6058.986,E2 6058.986} C_VEL
LIN {X 0,Y 97.04,Z 1065.183,A -85,B 0,C 180,E1 6047.386,E2 6047.386} C_VEL
LIN {X 0,Y 96.007,Z 1065.973,A -85,B 0,C 180,E1 6035.978,E2 6035.978} C_VEL
LIN {X 0,Y 96.048,Z 1065.87,A -85,B 0,C 180,E1 6028.21,E2 6028.21} C_VEL
LIN {X 0,Y 96.117,Z 1065.222,A -85,B 0,C 180,E1 6019.814,E2 6019.814} C_VEL
LIN {X 0,Y 97.878,Z 1063.551,A -85,B 0,C 180,E1 6009.05,E2 6009.05} C_VEL
LIN {X 0,Y 103.223,Z 1060.462,A -85,B 0,C 180,E1 5997.149,E2 5997.149} C_VEL
LIN {X 0,Y 114.077,Z 1055.067,A -85,B 0,C 180,E1 5984.768,E2 5984.768} C_VEL
LIN {X 0,Y 126.363,Z 1049.078,A -85,B 0,C 180,E1 5976.186,E2 5976.186} C_VEL
LIN {X 0,Y 143.055,Z 1040.576,A -85,B 0,C 180,E1 5968.275,E2 5968.275} C_VEL
LIN {X 0,Y 159.38,Z 1031.449,A -85,B 0,C 180,E1 5962.747,E2 5962.747} C_VEL
LIN {X 0,Y 178.099,Z 1020.059,A -85,B 0,C 180,E1 5957.986,E2 5957.986} C_VEL
LIN {X 0,Y 196.16,Z 1007.623,A -85,B 0,C 180,E1 5954.422,E2 5954.422} C_VEL
LIN {X 0,Y 214.315,Z 993.867,A -85,B 0,C 180,E1 5951.549,E2 5951.549} C_VEL
LIN {X 0,Y 231.985,Z 978.69,A -85,B 0,C 180,E1 5949.24,E2 5949.24} C_VEL
LIN {X 0,Y 247.121,Z 964.299,A -85,B 0,C 180,E1 5947.56,E2 5947.56} C_VEL
LIN {X 0,Y 265.341,Z 944.789,A -85,B 0,C 180,E1 5945.826,E2 5945.826} C_VEL
LIN {X 0,Y 278.906,Z 928.369,A -85,B 0,C 180,E1 5944.697,E2 5944.697} C_VEL
LIN {X 0,Y 294.013,Z 907.779,A -85,B 0,C 180,E1 5943.593,E2 5943.593} C_VEL
LIN {X 0,Y 306.326,Z 888.461,A -85,B 0,C 180,E1 5942.779,E2 5942.779} C_VEL
LIN {X 0,Y 318.432,Z 866.87,A -85,B 0,C 180,E1 5942.064,E2 5942.064} C_VEL
LIN {X 0,Y 328.577,Z 845.349,A -85,B 0,C 180,E1 5941.509,E2 5941.509} C_VEL
LIN {X 0,Y 337.52,Z 823.187,A -85,B 0,C 180,E1 5941.06,E2 5941.06} C_VEL
LIN {X 0,Y 345.393,Z 798.893,A -85,B 0,C 180,E1 5940.69,E2 5940.69} C_VEL
LIN {X 0,Y 351.22,Z 776.228,A -85,B 0,C 180,E1 5940.412,E2 5940.412} C_VEL
LIN {X 0,Y 355.924,Z 750.691,A -85,B 0,C 180,E1 5940.118,E2 5940.118} C_VEL
LIN {X 0,Y 365.441,Z 674.378,A -85,B 0,C 180,E1 5939.268,E2 5939.268} C_VEL
LIN {X 0,Y 365.453,Z 674.197,A -85,B 0,C 180,E1 5938.589,E2 5938.589} C_VEL
LIN {X 0,Y 365.423,Z 674.503,A -85,B 0,C 180,E1 5938.357,E2 5938.357} C_VEL
LIN {X 0,Y 355.505,Z 753.47,A -85,B 0,C 180,E1 5937.49,E2 5937.49} C_VEL
LIN {X 0,Y 350.522,Z 778.873,A -85,B 0,C 180,E1 5937.184,E2 5937.184} C_VEL
LIN {X 0,Y 344.792,Z 800.65,A -85,B 0,C 180,E1 5936.861,E2 5936.861} C_VEL
LIN {X 0,Y 336.631,Z 825.054,A -85,B 0,C 180,E1 5936.39,E2 5936.39} C_VEL
LIN {X 0,Y 328.294,Z 845.491,A -85,B 0,C 180,E1 5935.886,E2 5935.886} C_VEL
LIN {X 0,Y 317.524,Z 867.951,A -85,B 0,C 180,E1 5935.203,E2 5935.203} C_VEL
LIN {X 0,Y 305.914,Z 888.421,A -85,B 0,C 180,E1 5934.423,E2 5934.423} C_VEL
LIN {X 0,Y 292.385,Z 909.331,A -85,B 0,C 180,E1 5933.435,E2 5933.435} C_VEL
LIN {X 0,Y 277.993,Z 928.505,A -85,B 0,C 180,E1 5932.273,E2 5932.273} C_VEL
LIN {X 0,Y 262.306,Z 947.137,A -85,B 0,C 180,E1 5930.854,E2 5930.854} C_VEL
LIN {X 0,Y 245.389,Z 964.604,A -85,B 0,C 180,E1 5929.114,E2 5929.114} C_VEL
LIN {X 0,Y 227.81,Z 980.892,A -85,B 0,C 180,E1 5927.004,E2 5927.004} C_VEL
LIN {X 0,Y 209.677,Z 995.591,A -85,B 0,C 180,E1 5924.425,E2 5924.425} C_VEL
LIN {X 0,Y 191.171,Z 1009.129,A -85,B 0,C 180,E1 5921.207,E2 5921.207} C_VEL
LIN {X 0,Y 172.586,Z 1021.044,A -85,B 0,C 180,E1 5917.159,E2 5917.159} C_VEL
LIN {X 0,Y 154.901,Z 1031.369,A -85,B 0,C 180,E1 5912.17,E2 5912.17} C_VEL
LIN {X 0,Y 137.923,Z 1040.139,A -85,B 0,C 180,E1 5905.736,E2 5905.736} C_VEL
LIN {X 0,Y 122.978,Z 1047.366,A -85,B 0,C 180,E1 5897.722,E2 5897.722} C_VEL
LIN {X 0,Y 110.299,Z 1053.09,A -85,B 0,C 180,E1 5887.399,E2 5887.399} C_VEL
LIN {X 0,Y 102.317,Z 1056.798,A -85,B 0,C 180,E1 5876.714,E2 5876.714} C_VEL
LIN {X 0,Y 97.271,Z 1059.603,A -85,B 0,C 180,E1 5863.07,E2 5863.07} C_VEL
LIN {X 0,Y 96.111,Z 1060.667,A -85,B 0,C 180,E1 5851.788,E2 5851.788} C_VEL
LIN {X 0,Y 96.193,Z 1060.888,A -85,B 0,C 180,E1 5842.234,E2 5842.234} C_VEL
LIN {X 0,Y 97.763,Z 1060.262,A -85,B 0,C 180,E1 5830.896,E2 5830.896} C_VEL
LIN {X 0,Y 102.316,Z 1058.578,A -85,B 0,C 180,E1 5819.458,E2 5819.458} C_VEL
LIN {X 0,Y 111.891,Z 1055.195,A -85,B 0,C 180,E1 5807.222,E2 5807.222} C_VEL
LIN {X 0,Y 125.302,Z 1049.99,A -85,B 0,C 180,E1 5797.062,E2 5797.062} C_VEL
LIN {X 0,Y 141.681,Z 1043.231,A -85,B 0,C 180,E1 5788.942,E2 5788.942} C_VEL
LIN {X 0,Y 159.386,Z 1034.846,A -85,B 0,C 180,E1 5782.752,E2 5782.752} C_VEL
LIN {X 0,Y 177.673,Z 1025.286,A -85,B 0,C 180,E1 5777.996,E2 5777.996} C_VEL
LIN {X 0,Y 196.95,Z 1013.725,A -85,B 0,C 180,E1 5774.105,E2 5774.105} C_VEL
LIN {X 0,Y 215.062,Z 1001.627,A -85,B 0,C 180,E1 5771.186,E2 5771.186} C_VEL
LIN {X 0,Y 233.668,Z 987.512,A -85,B 0,C 180,E1 5768.707,E2 5768.707} C_VEL
LIN {X 0,Y 249.776,Z 973.849,A -85,B 0,C 180,E1 5766.888,E2 5766.888} C_VEL
LIN {X 0,Y 268.521,Z 955.929,A -85,B 0,C 180,E1 5765.069,E2 5765.069} C_VEL
LIN {X 0,Y 283.591,Z 939.584,A -85,B 0,C 180,E1 5763.795,E2 5763.795} C_VEL
LIN {X 0,Y 299.769,Z 919.763,A -85,B 0,C 180,E1 5762.572,E2 5762.572} C_VEL
LIN {X 0,Y 312.603,Z 901.752,A -85,B 0,C 180,E1 5761.699,E2 5761.699} C_VEL
LIN {X 0,Y 325.766,Z 880.868,A -85,B 0,C 180,E1 5760.879,E2 5760.879} C_VEL
LIN {X 0,Y 336.965,Z 859.912,A -85,B 0,C 180,E1 5760.214,E2 5760.214} C_VEL
LIN {X 0,Y 346.968,Z 838.28,A -85,B 0,C 180,E1 5759.668,E2 5759.668} C_VEL
LIN {X 0,Y 355.544,Z 815.784,A -85,B 0,C 180,E1 5759.219,E2 5759.219} C_VEL
LIN {X 0,Y 355.996,Z 814.447,A -85,B 0,C 180,E1 5759.188,E2 5759.188} C_VEL
LIN {X 0,Y 347.584,Z 836.962,A -85,B 0,C 180,E1 5758.831,E2 5758.831} C_VEL
LIN {X 0,Y 337.598,Z 858.809,A -85,B 0,C 180,E1 5758.379,E2 5758.379} C_VEL
LIN {X 0,Y 326.699,Z 879.453,A -85,B 0,C 180,E1 5757.826,E2 5757.826} C_VEL
LIN {X 0,Y 313.371,Z 901.034,A -85,B 0,C 180,E1 5757.087,E2 5757.087} C_VEL
LIN {X 0,Y 300.592,Z 919.194,A -85,B 0,C 180,E1 5756.303,E2 5756.303} C_VEL
LIN {X 0,Y 283.805,Z 940.086,A -85,B 0,C 180,E1 5755.15,E2 5755.15} C_VEL
LIN {X 0,Y 268.954,Z 956.383,A -85,B 0,C 180,E1 5753.979,E2 5753.979} C_VEL
LIN {X 0,Y 250.243,Z 974.596,A -85,B 0,C 180,E1 5752.276,E2 5752.276} C_VEL
LIN {X 0,Y 249.133,Z 975.585,A -85,B 0,C 180,E1 5752.165,E2 5752.165} C_VEL
LIN {X 0,Y 243.335,Z 980.639,A -85,B 0,C 180,E1 5751.824,E2 5751.824} C_VEL
LIN {X 0,Y 226.543,Z 993.596,A -85,B 0,C 180,E1 5751.646,E2 5751.646} C_VEL
LIN {X 0,Y 221.35,Z 997.366,A -85,B 0,C 180,E1 5751.254,E2 5751.254} C_VEL
LIN {X 0,Y 202.819,Z 1010.504,A -85,B 0,C 180,E1 5748.832,E2 5748.832} C_VEL
LIN {X 0,Y 182.748,Z 1022.98,A -85,B 0,C 180,E1 5745.567,E2 5745.567} C_VEL
LIN {X 0,Y 165.138,Z 1032.771,A -85,B 0,C 180,E1 5741.918,E2 5741.918} C_VEL
LIN {X 0,Y 144.307,Z 1042.999,A -85,B 0,C 180,E1 5736.151,E2 5736.151} C_VEL
LIN {X 0,Y 127.501,Z 1050.331,A -85,B 0,C 180,E1 5729.615,E2 5729.615} C_VEL
LIN {X 0,Y 110.313,Z 1057.079,A -85,B 0,C 180,E1 5719.586,E2 5719.586} C_VEL
LIN {X 0,Y 98.962,Z 1061.257,A -85,B 0,C 180,E1 5708.788,E2 5708.788} C_VEL
LIN {X 0,Y 90.63,Z 1064.429,A -85,B 0,C 180,E1 5693.693,E2 5693.693} C_VEL
LIN {X 0,Y 88.134,Z 1065.603,A -85,B 0,C 180,E1 5680.458,E2 5680.458} C_VEL
LIN {X 0,Y 88.052,Z 1065.765,A -85,B 0,C 180,E1 5671.301,E2 5671.301} C_VEL
LIN {X 0,Y 88.023,Z 1065.425,A -85,B 0,C 180,E1 5662.822,E2 5662.822} C_VEL
LIN {X 0,Y 89.748,Z 1063.674,A -85,B 0,C 180,E1 5649.114,E2 5649.114} C_VEL
LIN {X 0,Y 95.301,Z 1060.719,A -85,B 0,C 180,E1 5636.216,E2 5636.216} C_VEL
LIN {X 0,Y 106.474,Z 1055.721,A -85,B 0,C 180,E1 5623.278,E2 5623.278} C_VEL
LIN {X 0,Y 120.287,Z 1049.437,A -85,B 0,C 180,E1 5613.773,E2 5613.773} C_VEL
LIN {X 0,Y 136.984,Z 1041.509,A -85,B 0,C 180,E1 5606.128,E2 5606.128} C_VEL
LIN {X 0,Y 155.517,Z 1031.63,A -85,B 0,C 180,E1 5600.166,E2 5600.166} C_VEL
LIN {X 0,Y 173.581,Z 1021.061,A -85,B 0,C 180,E1 5595.85,E2 5595.85} C_VEL
LIN {X 0,Y 192.966,Z 1008.226,A -85,B 0,C 180,E1 5592.266,E2 5592.266} C_VEL
LIN {X 0,Y 210.003,Z 995.679,A -85,B 0,C 180,E1 5589.738,E2 5589.738} C_VEL
LIN {X 0,Y 229.85,Z 979.204,A -85,B 0,C 180,E1 5587.324,E2 5587.324} C_VEL
LIN {X 0,Y 246.174,Z 963.947,A -85,B 0,C 180,E1 5585.663,E2 5585.663} C_VEL
LIN {X 0,Y 263.748,Z 945.429,A -85,B 0,C 180,E1 5584.131,E2 5584.131} C_VEL
LIN {X 0,Y 277.864,Z 928.591,A -85,B 0,C 180,E1 5583.054,E2 5583.054} C_VEL
LIN {X 0,Y 292.658,Z 908.786,A -85,B 0,C 180,E1 5582.066,E2 5582.066} C_VEL
LIN {X 0,Y 305.543,Z 888.83,A -85,B 0,C 180,E1 5581.286,E2 5581.286} C_VEL
LIN {X 0,Y 317.485,Z 867.823,A -85,B 0,C 180,E1 5580.642,E2 5580.642} C_VEL
LIN {X 0,Y 327.964,Z 845.95,A -85,B 0,C 180,E1 5580.121,E2 5580.121} C_VEL
LIN {X 0,Y 336.413,Z 825.329,A -85,B 0,C 180,E1 5579.732,E2 5579.732} C_VEL
LIN {X 0,Y 344.92,Z 799.821,A -85,B 0,C 180,E1 5579.371,E2 5579.371} C_VEL
LIN {X 0,Y 350.663,Z 777.892,A -85,B 0,C 180,E1 5579.123,E2 5579.123} C_VEL
LIN {X 0,Y 355.751,Z 751.195,A -85,B 0,C 180,E1 5578.832,E2 5578.832} C_VEL
LIN {X 0,Y 355.871,Z 750.371,A -85,B 0,C 180,E1 5578.815,E2 5578.815} C_VEL
LIN {X 0,Y 351.138,Z 775.853,A -85,B 0,C 180,E1 5578.535,E2 5578.535} C_VEL
LIN {X 0,Y 345.293,Z 798.416,A -85,B 0,C 180,E1 5578.231,E2 5578.231} C_VEL
LIN {X 0,Y 337.707,Z 821.809,A -85,B 0,C 180,E1 5577.822,E2 5577.822} C_VEL
LIN {X 0,Y 328.819,Z 843.752,A -85,B 0,C 180,E1 5577.335,E2 5577.335} C_VEL
LIN {X 0,Y 318.916,Z 864.668,A -85,B 0,C 180,E1 5576.765,E2 5576.765} C_VEL
LIN {X 0,Y 306.707,Z 886.457,A -85,B 0,C 180,E1 5576.015,E2 5576.015} C_VEL
LIN {X 0,Y 294.496,Z 905.464,A -85,B 0,C 180,E1 5575.21,E2 5575.21} C_VEL
LIN {X 0,Y 278.96,Z 926.488,A -85,B 0,C 180,E1 5574.074,E2 5574.074} C_VEL
LIN {X 0,Y 264.982,Z 943.141,A -85,B 0,C 180,E1 5572.936,E2 5572.936} C_VEL
LIN {X 0,Y 246.837,Z 962.211,A -85,B 0,C 180,E1 5571.264,E2 5571.264} C_VEL
LIN {X 0,Y 231.737,Z 976.253,A -85,B 0,C 180,E1 5569.661,E2 5569.661} C_VEL
LIN {X 0,Y 213.152,Z 991.768,A -85,B 0,C 180,E1 5567.348,E2 5567.348} C_VEL
LIN {X 0,Y 194.957,Z 1005.081,A -85,B 0,C 180,E1 5564.624,E2 5564.624} C_VEL
LIN {X 0,Y 176.117,Z 1017.5,A -85,B 0,C 180,E1 5561.118,E2 5561.118} C_VEL
LIN {X 0,Y 157.776,Z 1028.058,A -85,B 0,C 180,E1 5556.769,E2 5556.769} C_VEL
LIN {X 0,Y 140.261,Z 1037.215,A -85,B 0,C 180,E1 5551.264,E2 5551.264} C_VEL
LIN {X 0,Y 122.904,Z 1045.263,A -85,B 0,C 180,E1 5543.651,E2 5543.651} C_VEL
LIN {X 0,Y 109.249,Z 1051.162,A -85,B 0,C 180,E1 5534.808,E2 5534.808} C_VEL
LIN {X 0,Y 97.328,Z 1056.113,A -85,B 0,C 180,E1 5522.291,E2 5522.291} C_VEL
LIN {X 0,Y 91.023,Z 1058.925,A -85,B 0,C 180,E1 5509.909,E2 5509.909} C_VEL
LIN {X 0,Y 88.453,Z 1060.477,A -85,B 0,C 180,E1 5497.796,E2 5497.796} C_VEL
LIN {X 0,Y 88.054,Z 1061.026,A -85,B 0,C 180,E1 5487.835,E2 5487.835} C_VEL
LIN {X 0,Y 88.473,Z 1061.001,A -85,B 0,C 180,E1 5478.262,E2 5478.262} C_VEL
LIN {X 0,Y 91.091,Z 1060.152,A -85,B 0,C 180,E1 5466.037,E2 5466.037} C_VEL
LIN {X 0,Y 99.237,Z 1057.566,A -85,B 0,C 180,E1 5451.34,E2 5451.34} C_VEL
LIN {X 0,Y 110.436,Z 1053.779,A -85,B 0,C 180,E1 5440.488,E2 5440.488} C_VEL
LIN {X 0,Y 126.018,Z 1048.173,A -85,B 0,C 180,E1 5431.026,E2 5431.026} C_VEL
LIN {X 0,Y 143.827,Z 1040.75,A -85,B 0,C 180,E1 5423.78,E2 5423.78} C_VEL
LIN {X 0,Y 163.131,Z 1031.79,A -85,B 0,C 180,E1 5418.185,E2 5418.185} C_VEL
LIN {X 0,Y 182.729,Z 1021.212,A -85,B 0,C 180,E1 5413.932,E2 5413.932} C_VEL
LIN {X 0,Y 202.435,Z 1009.317,A -85,B 0,C 180,E1 5410.604,E2 5410.604} C_VEL
LIN {X 0,Y 221.152,Z 996.301,A -85,B 0,C 180,E1 5408.044,E2 5408.044} C_VEL
LIN {X 0,Y 239.277,Z 982.251,A -85,B 0,C 180,E1 5405.984,E2 5405.984} C_VEL
LIN {X 0,Y 257.666,Z 965.973,A -85,B 0,C 180,E1 5404.206,E2 5404.206} C_VEL
LIN {X 0,Y 273.319,Z 950.438,A -85,B 0,C 180,E1 5402.894,E2 5402.894} C_VEL
LIN {X 0,Y 290.584,Z 930.957,A -85,B 0,C 180,E1 5401.617,E2 5401.617} C_VEL
LIN {X 0,Y 303.991,Z 913.78,A -85,B 0,C 180,E1 5400.725,E2 5400.725} C_VEL
LIN {X 0,Y 318.966,Z 891.862,A -85,B 0,C 180,E1 5399.828,E2 5399.828} C_VEL
LIN {X 0,Y 328.112,Z 876.569,A -85,B 0,C 180,E1 5399.319,E2 5399.319} C_VEL
LIN {X 0,Y 314.057,Z 899.556,A -85,B 0,C 180,E1 5398.618,E2 5398.618} C_VEL
LIN {X 0,Y 301.168,Z 917.831,A -85,B 0,C 180,E1 5397.907,E2 5397.907} C_VEL
LIN {X 0,Y 284.882,Z 938.162,A -85,B 0,C 180,E1 5396.9,E2 5396.9} C_VEL
LIN {X 0,Y 269.198,Z 955.294,A -85,B 0,C 180,E1 5395.787,E2 5395.787} C_VEL
LIN {X 0,Y 251.21,Z 972.801,A -85,B 0,C 180,E1 5394.311,E2 5394.311} C_VEL
LIN {X 0,Y 233.664,Z 987.783,A -85,B 0,C 180,E1 5392.624,E2 5392.624} C_VEL
LIN {X 0,Y 221.35,Z 997.366,A -85,B 0,C 180,E1 5391.254,E2 5391.254} C_VEL
LIN {X 0,Y 215.178,Z 1001.856,A -85,B 0,C 180,E1 5390.79,E2 5390.79} C_VEL
LIN {X 0,Y 197.26,Z 1013.111,A -85,B 0,C 180,E1 5390.347,E2 5390.347} C_VEL
LIN {X 0,Y 191.799,Z 1016.363,A -85,B 0,C 180,E1 5389.815,E2 5389.815} C_VEL
LIN {X 0,Y 170.831,Z 1028.435,A -85,B 0,C 180,E1 5386.315,E2 5386.315} C_VEL
LIN {X 0,Y 152.223,Z 1037.766,A -85,B 0,C 180,E1 5382.259,E2 5382.259} C_VEL
LIN {X 0,Y 132.598,Z 1046.572,A -85,B 0,C 180,E1 5376.443,E2 5376.443} C_VEL
LIN {X 0,Y 114.639,Z 1053.495,A -85,B 0,C 180,E1 5368.734,E2 5368.734} C_VEL
LIN {X 0,Y 99.066,Z 1059.019,A -85,B 0,C 180,E1 5358.322,E2 5358.322} C_VEL
LIN {X 0,Y 87.485,Z 1062.753,A -85,B 0,C 180,E1 5344.853,E2 5344.853} C_VEL
LIN {X 0,Y 81.821,Z 1064.694,A -85,B 0,C 180,E1 5331.507,E2 5331.507} C_VEL
LIN {X 0,Y 80.039,Z 1065.524,A -85,B 0,C 180,E1 5317.899,E2 5317.899} C_VEL
LIN {X 0,Y 80.065,Z 1065.483,A -85,B 0,C 180,E1 5309.285,E2 5309.285} C_VEL
LIN {X 0,Y 80.143,Z 1064.915,A -85,B 0,C 180,E1 5299.214,E2 5299.214} C_VEL
LIN {X 0,Y 82.601,Z 1063.202,A -85,B 0,C 180,E1 5285.696,E2 5285.696} C_VEL
LIN {X 0,Y 89.405,Z 1060.143,A -85,B 0,C 180,E1 5272.04,E2 5272.04} C_VEL
LIN {X 0,Y 103.092,Z 1054.553,A -85,B 0,C 180,E1 5258.222,E2 5258.222} C_VEL
LIN {X 0,Y 117.353,Z 1048.538,A -85,B 0,C 180,E1 5249.616,E2 5249.616} C_VEL
LIN {X 0,Y 136.792,Z 1039.602,A -85,B 0,C 180,E1 5241.827,E2 5241.827} C_VEL
LIN {X 0,Y 154.592,Z 1030.405,A -85,B 0,C 180,E1 5236.813,E2 5236.813} C_VEL
LIN {X 0,Y 175.138,Z 1018.524,A -85,B 0,C 180,E1 5232.509,E2 5232.509} C_VEL
LIN {X 0,Y 192.704,Z 1006.997,A -85,B 0,C 180,E1 5229.647,E2 5229.647} C_VEL
LIN {X 0,Y 211.627,Z 993.223,A -85,B 0,C 180,E1 5227.16,E2 5227.16} C_VEL
LIN {X 0,Y 229.914,Z 978.005,A -85,B 0,C 180,E1 5225.18,E2 5225.18} C_VEL
LIN {X 0,Y 246.479,Z 962.656,A -85,B 0,C 180,E1 5223.672,E2 5223.672} C_VEL
LIN {X 0,Y 264.181,Z 944.031,A -85,B 0,C 180,E1 5222.285,E2 5222.285} C_VEL
LIN {X 0,Y 278.388,Z 927.159,A -85,B 0,C 180,E1 5221.315,E2 5221.315} C_VEL
LIN {X 0,Y 294.473,Z 905.391,A -85,B 0,C 180,E1 5220.355,E2 5220.355} C_VEL
LIN {X 0,Y 306.513,Z 886.674,A -85,B 0,C 180,E1 5219.705,E2 5219.705} C_VEL
LIN {X 0,Y 319.052,Z 864.267,A -85,B 0,C 180,E1 5219.102,E2 5219.102} C_VEL
LIN {X 0,Y 328.048,Z 845.409,A -85,B 0,C 180,E1 5218.702,E2 5218.702} C_VEL
LIN {X 0,Y 317.135,Z 867.907,A -85,B 0,C 180,E1 5218.123,E2 5218.123} C_VEL
LIN {X 0,Y 305.267,Z 888.511,A -85,B 0,C 180,E1 5217.455,E2 5217.455} C_VEL
LIN {X 0,Y 291.969,Z 908.796,A -85,B 0,C 180,E1 5216.644,E2 5216.644} C_VEL
LIN {X 0,Y 277.285,Z 928.057,A -85,B 0,C 180,E1 5215.657,E2 5215.657} C_VEL
LIN {X 0,Y 262.321,Z 945.54,A -85,B 0,C 180,E1 5214.532,E2 5214.532} C_VEL
LIN {X 0,Y 244.776,Z 963.475,A -85,B 0,C 180,E1 5213.042,E2 5213.042} C_VEL
LIN {X 0,Y 228.518,Z 978.259,A -85,B 0,C 180,E1 5211.444,E2 5211.444} C_VEL
LIN {X 0,Y 208.712,Z 994.157,A -85,B 0,C 180,E1 5209.145,E2 5209.145} C_VEL
LIN {X 0,Y 191.334,Z 1006.498,A -85,B 0,C 180,E1 5206.706,E2 5206.706} C_VEL
LIN {X 0,Y 170.399,Z 1019.643,A -85,B 0,C 180,E1 5203.033,E2 5203.033} C_VEL
LIN {X 0,Y 153.038,Z 1029.242,A -85,B 0,C 180,E1 5199.116,E2 5199.116} C_VEL
LIN {X 0,Y 133.346,Z 1038.953,A -85,B 0,C 180,E1 5193.166,E2 5193.166} C_VEL
LIN {X 0,Y 116.827,Z 1046.116,A -85,B 0,C 180,E1 5186.118,E2 5186.118} C_VEL
LIN {X 0,Y 101.262,Z 1052.384,A -85,B 0,C 180,E1 5176.122,E2 5176.122} C_VEL
LIN {X 0,Y 89.323,Z 1056.815,A -85,B 0,C 180,E1 5163.265,E2 5163.265} C_VEL
LIN {X 0,Y 82.695,Z 1059.54,A -85,B 0,C 180,E1 5149.417,E2 5149.417} C_VEL
LIN {X 0,Y 80.2,Z 1061.036,A -85,B 0,C 180,E1 5134.29,E2 5134.29} C_VEL
LIN {X 0,Y 80.106,Z 1061.354,A -85,B 0,C 180,E1 5124.269,E2 5124.269} C_VEL
LIN {X 0,Y 81.637,Z 1060.995,A -85,B 0,C 180,E1 5110.689,E2 5110.689} C_VEL
LIN {X 0,Y 87.429,Z 1059.308,A -85,B 0,C 180,E1 5095.917,E2 5095.917} C_VEL
LIN {X 0,Y 97.026,Z 1056.529,A -85,B 0,C 180,E1 5083.831,E2 5083.831} C_VEL
LIN {X 0,Y 113.467,Z 1051.27,A -85,B 0,C 180,E1 5071.92,E2 5071.92} C_VEL
LIN {X 0,Y 129.65,Z 1045.379,A -85,B 0,C 180,E1 5064.488,E2 5064.488} C_VEL
LIN {X 0,Y 150.284,Z 1036.767,A -85,B 0,C 180,E1 5057.931,E2 5057.931} C_VEL
LIN {X 0,Y 168.755,Z 1027.861,A -85,B 0,C 180,E1 5053.66,E2 5053.66} C_VEL
LIN {X 0,Y 189.82,Z 1016.29,A -85,B 0,C 180,E1 5049.925,E2 5049.925} C_VEL
LIN {X 0,Y 208.661,Z 1004.403,A -85,B 0,C 180,E1 5047.285,E2 5047.285} C_VEL
LIN {X 0,Y 228.838,Z 990.026,A -85,B 0,C 180,E1 5044.979,E2 5044.979} C_VEL
LIN {X 0,Y 246.38,Z 975.724,A -85,B 0,C 180,E1 5043.294,E2 5043.294} C_VEL
LIN {X 0,Y 264.601,Z 959.103,A -85,B 0,C 180,E1 5041.8,E2 5041.8} C_VEL
LIN {X 0,Y 281.179,Z 941.699,A -85,B 0,C 180,E1 5040.611,E2 5040.611} C_VEL
LIN {X 0,Y 296.878,Z 923.215,A -85,B 0,C 180,E1 5039.614,E2 5039.614} C_VEL
LIN {X 0,Y 300.211,Z 918.838,A -85,B 0,C 180,E1 5039.411,E2 5039.411} C_VEL
LIN {X 0,Y 283.073,Z 939.768,A -85,B 0,C 180,E1 5038.447,E2 5038.447} C_VEL
LIN {X 0,Y 268.228,Z 955.73,A -85,B 0,C 180,E1 5037.488,E2 5037.488} C_VEL
LIN {X 0,Y 249.527,Z 973.574,A -85,B 0,C 180,E1 5036.094,E2 5036.094} C_VEL
LIN {X 0,Y 232.02,Z 988.26,A -85,B 0,C 180,E1 5034.559,E2 5034.559} C_VEL
LIN {X 0,Y 212.779,Z 1002.699,A -85,B 0,C 180,E1 5032.537,E2 5032.537} C_VEL
LIN {X 0,Y 192.923,Z 1015.667,A -85,B 0,C 180,E1 5029.978,E2 5029.978} C_VEL
LIN {X 0,Y 191.799,Z 1016.363,A -85,B 0,C 180,E1 5029.815,E2 5029.815} C_VEL
LIN {X 0,Y 185.333,Z 1020.186,A -85,B 0,C 180,E1 5029.175,E2 5029.175} C_VEL
LIN {X 0,Y 167.502,Z 1029.198,A -85,B 0,C 180,E1 5028.389,E2 5028.389} C_VEL
LIN {X 0,Y 160.882,Z 1032.406,A -85,B 0,C 180,E1 5027.557,E2 5027.557} C_VEL
LIN {X 0,Y 139.306,Z 1042.3,A -85,B 0,C 180,E1 5022.674,E2 5022.674} C_VEL
LIN {X 0,Y 121.592,Z 1049.357,A -85,B 0,C 180,E1 5017.074,E2 5017.074} C_VEL
LIN {X 0,Y 102.483,Z 1056.058,A -85,B 0,C 180,E1 5008.085,E2 5008.085} C_VEL
LIN {X 0,Y 87.831,Z 1060.53,A -85,B 0,C 180,E1 4996.769,E2 4996.769} C_VEL
LIN {X 0,Y 76.857,Z 1063.792,A -85,B 0,C 180,E1 4980.835,E2 4980.835} C_VEL
LIN {X 0,Y 72.357,Z 1065.15,A -85,B 0,C 180,E1 4963.587,E2 4963.587} C_VEL
LIN {X 0,Y 72.042,Z 1065.346,A -85,B 0,C 180,E1 4952.121,E2 4952.121} C_VEL
LIN {X 0,Y 72.025,Z 1065.072,A -85,B 0,C 180,E1 4942.823,E2 4942.823} C_VEL
LIN {X 0,Y 74.261,Z 1063.444,A -85,B 0,C 180,E1 4926.176,E2 4926.176} C_VEL
LIN {X 0,Y 81.233,Z 1060.567,A -85,B 0,C 180,E1 4911.116,E2 4911.116} C_VEL
LIN {X 0,Y 93.633,Z 1056.048,A -85,B 0,C 180,E1 4897.793,E2 4897.793} C_VEL
LIN {X 0,Y 110.388,Z 1049.53,A -85,B 0,C 180,E1 4887.417,E2 4887.417} C_VEL
LIN {X 0,Y 127.162,Z 1042.412,A -85,B 0,C 180,E1 4880.657,E2 4880.657} C_VEL
LIN {X 0,Y 147.917,Z 1032.458,A -85,B 0,C 180,E1 4874.838,E2 4874.838} C_VEL
LIN {X 0,Y 166.091,Z 1022.567,A -85,B 0,C 180,E1 4871.104,E2 4871.104} C_VEL
LIN {X 0,Y 186.728,Z 1009.912,A -85,B 0,C 180,E1 4867.847,E2 4867.847} C_VEL
LIN {X 0,Y 204.943,Z 997.17,A -85,B 0,C 180,E1 4865.563,E2 4865.563} C_VEL
LIN {X 0,Y 224.412,Z 981.948,A -85,B 0,C 180,E1 4863.575,E2 4863.575} C_VEL
LIN {X 0,Y 242.13,Z 966.054,A -85,B 0,C 180,E1 4862.063,E2 4862.063} C_VEL
LIN {X 0,Y 258.999,Z 949.173,A -85,B 0,C 180,E1 4860.837,E2 4860.837} C_VEL
LIN {X 0,Y 275.526,Z 930.197,A -85,B 0,C 180,E1 4859.792,E2 4859.792} C_VEL
LIN {X 0,Y 290.012,Z 911.432,A -85,B 0,C 180,E1 4859,E2 4859} C_VEL
LIN {X 0,Y 298.058,Z 899.767,A -85,B 0,C 180,E1 4858.583,E2 4858.583} C_VEL
LIN {X 0,Y 285.17,Z 917.82,A -85,B 0,C 180,E1 4857.843,E2 4857.843} C_VEL
LIN {X 0,Y 268.398,Z 938.404,A -85,B 0,C 180,E1 4856.763,E2 4856.763} C_VEL
LIN {X 0,Y 253.642,Z 954.276,A -85,B 0,C 180,E1 4855.704,E2 4855.704} C_VEL
LIN {X 0,Y 236.156,Z 971.092,A -85,B 0,C 180,E1 4854.265,E2 4854.265} C_VEL
LIN {X 0,Y 217.834,Z 986.434,A -85,B 0,C 180,E1 4852.51,E2 4852.51} C_VEL
LIN {X 0,Y 198.809,Z 1000.684,A -85,B 0,C 180,E1 4850.32,E2 4850.32} C_VEL
LIN {X 0,Y 179.193,Z 1013.415,A -85,B 0,C 180,E1 4847.551,E2 4847.551} C_VEL
LIN {X 0,Y 160.082,Z 1024.484,A -85,B 0,C 180,E1 4844.133,E2 4844.133} C_VEL
LIN {X 0,Y 139.935,Z 1034.598,A -85,B 0,C 180,E1 4839.398,E2 4839.398} C_VEL
LIN {X 0,Y 121.77,Z 1042.674,A -85,B 0,C 180,E1 4833.512,E2 4833.512} C_VEL
LIN {X 0,Y 103.085,Z 1049.94,A -85,B 0,C 180,E1 4824.564,E2 4824.564} C_VEL
LIN {X 0,Y 89.246,Z 1054.832,A -85,B 0,C 180,E1 4813.998,E2 4813.998} C_VEL
LIN {X 0,Y 77.576,Z 1058.844,A -85,B 0,C 180,E1 4797.646,E2 4797.646} C_VEL
LIN {X 0,Y 73.023,Z 1060.664,A -85,B 0,C 180,E1 4782.655,E2 4782.655} C_VEL
LIN {X 0,Y 72.103,Z 1061.361,A -85,B 0,C 180,E1 4770.794,E2 4770.794} C_VEL
LIN {X 0,Y 72.33,Z 1061.523,A -85,B 0,C 180,E1 4759.647,E2 4759.647} C_VEL
LIN {X 0,Y 75.099,Z 1060.884,A -85,B 0,C 180,E1 4744.782,E2 4744.782} C_VEL
LIN {X 0,Y 82.063,Z 1059.185,A -85,B 0,C 180,E1 4730.685,E2 4730.685} C_VEL
LIN {X 0,Y 95.205,Z 1055.765,A -85,B 0,C 180,E1 4717.042,E2 4717.042} C_VEL
LIN {X 0,Y 111.334,Z 1050.788,A -85,B 0,C 180,E1 4707.237,E2 4707.237} C_VEL
LIN {X 0,Y 129.769,Z 1044.367,A -85,B 0,C 180,E1 4699.944,E2 4699.944} C_VEL
LIN {X 0,Y 149.722,Z 1036.129,A -85,B 0,C 180,E1 4694.452,E2 4694.452} C_VEL
LIN {X 0,Y 168.842,Z 1027.108,A -85,B 0,C 180,E1 4690.562,E2 4690.562} C_VEL
LIN {X 0,Y 190.474,Z 1015.29,A -85,B 0,C 180,E1 4687.183,E2 4687.183} C_VEL
LIN {X 0,Y 208.745,Z 1003.9,A -85,B 0,C 180,E1 4684.917,E2 4684.917} C_VEL
LIN {X 0,Y 230.237,Z 988.599,A -85,B 0,C 180,E1 4682.737,E2 4682.737} C_VEL
LIN {X 0,Y 247.037,Z 974.977,A -85,B 0,C 180,E1 4681.307,E2 4681.307} C_VEL
LIN {X 0,Y 265.971,Z 957.657,A -85,B 0,C 180,E1 4679.922,E2 4679.922} C_VEL
LIN {X 0,Y 272.432,Z 951.134,A -85,B 0,C 180,E1 4679.498,E2 4679.498} C_VEL
LIN {X 0,Y 257.057,Z 966.234,A -85,B 0,C 180,E1 4678.525,E2 4678.525} C_VEL
LIN {X 0,Y 238.269,Z 982.731,A -85,B 0,C 180,E1 4677.146,E2 4677.146} C_VEL
LIN {X 0,Y 219.646,Z 996.988,A -85,B 0,C 180,E1 4675.522,E2 4675.522} C_VEL
LIN {X 0,Y 199.577,Z 1010.714,A -85,B 0,C 180,E1 4673.383,E2 4673.383} C_VEL
LIN {X 0,Y 179.344,Z 1022.688,A -85,B 0,C 180,E1 4670.689,E2 4670.689} C_VEL
LIN {X 0,Y 160.882,Z 1032.406,A -85,B 0,C 180,E1 4667.557,E2 4667.557} C_VEL
LIN {X 0,Y 154.222,Z 1035.534,A -85,B 0,C 180,E1 4666.64,E2 4666.64} C_VEL
LIN {X 0,Y 135.788,Z 1042.77,A -85,B 0,C 180,E1 4665.192,E2 4665.192} C_VEL
LIN {X 0,Y 129.077,Z 1045.346,A -85,B 0,C 180,E1 4663.936,E2 4663.936} C_VEL
LIN {X 0,Y 108.601,Z 1052.605,A -85,B 0,C 180,E1 4657.029,E2 4657.029} C_VEL
LIN {X 0,Y 91.731,Z 1057.785,A -85,B 0,C 180,E1 4648.236,E2 4648.236} C_VEL
LIN {X 0,Y 75.353,Z 1062.165,A -85,B 0,C 180,E1 4633.129,E2 4633.129} C_VEL
LIN {X 0,Y 67.182,Z 1064.204,A -85,B 0,C 180,E1 4617.476,E2 4617.476} C_VEL
LIN {X 0,Y 64.136,Z 1065.073,A -85,B 0,C 180,E1 4600.783,E2 4600.783} C_VEL
LIN {X 0,Y 64.078,Z 1065.072,A -85,B 0,C 180,E1 4590,E2 4590} C_VEL
LIN {X 0,Y 64.18,Z 1064.608,A -85,B 0,C 180,E1 4578.315,E2 4578.315} C_VEL
LIN {X 0,Y 67.723,Z 1062.853,A -85,B 0,C 180,E1 4560.842,E2 4560.842} C_VEL
LIN {X 0,Y 76.546,Z 1059.824,A -85,B 0,C 180,E1 4545.14,E2 4545.14} C_VEL
LIN {X 0,Y 93.029,Z 1054.3,A -85,B 0,C 180,E1 4530.7,E2 4530.7} C_VEL
LIN {X 0,Y 109.254,Z 1048.329,A -85,B 0,C 180,E1 4522.429,E2 4522.429} C_VEL
LIN {X 0,Y 129.746,Z 1039.869,A -85,B 0,C 180,E1 4515.568,E2 4515.568} C_VEL
LIN {X 0,Y 148.777,Z 1030.765,A -85,B 0,C 180,E1 4511.12,E2 4511.12} C_VEL
LIN {X 0,Y 169.446,Z 1019.647,A -85,B 0,C 180,E1 4507.54,E2 4507.54} C_VEL
LIN {X 0,Y 189.75,Z 1006.955,A -85,B 0,C 180,E1 4504.836,E2 4504.836} C_VEL
LIN {X 0,Y 208.238,Z 994.002,A -85,B 0,C 180,E1 4502.872,E2 4502.872} C_VEL
LIN {X 0,Y 228.02,Z 978.178,A -85,B 0,C 180,E1 4501.147,E2 4501.147} C_VEL
LIN {X 0,Y 243.973,Z 963.826,A -85,B 0,C 180,E1 4499.981,E2 4499.981} C_VEL
LIN {X 0,Y 262.527,Z 944.959,A -85,B 0,C 180,E1 4498.815,E2 4498.815} C_VEL
LIN {X 0,Y 268.064,Z 938.779,A -85,B 0,C 180,E1 4498.485,E2 4498.485} C_VEL
LIN {X 0,Y 252.856,Z 954.951,A -85,B 0,C 180,E1 4497.507,E2 4497.507} C_VEL
LIN {X 0,Y 234.503,Z 972.265,A -85,B 0,C 180,E1 4496.15,E2 4496.15} C_VEL
LIN {X 0,Y 216.926,Z 986.762,A -85,B 0,C 180,E1 4494.636,E2 4494.636} C_VEL
LIN {X 0,Y 197.604,Z 1000.999,A -85,B 0,C 180,E1 4492.645,E2 4492.645} C_VEL
LIN {X 0,Y 177.615,Z 1013.715,A -85,B 0,C 180,E1 4490.119,E2 4490.119} C_VEL
LIN {X 0,Y 158.047,Z 1024.777,A -85,B 0,C 180,E1 4486.978,E2 4486.978} C_VEL
LIN {X 0,Y 137.276,Z 1034.875,A -85,B 0,C 180,E1 4482.588,E2 4482.588} C_VEL
LIN {X 0,Y 118.356,Z 1042.943,A -85,B 0,C 180,E1 4477.05,E2 4477.05} C_VEL
LIN {X 0,Y 98.584,Z 1050.194,A -85,B 0,C 180,E1 4468.427,E2 4468.427} C_VEL
LIN {X 0,Y 83.59,Z 1055.079,A -85,B 0,C 180,E1 4457.87,E2 4457.87} C_VEL
LIN {X 0,Y 70.513,Z 1059.076,A -85,B 0,C 180,E1 4440.696,E2 4440.696} C_VEL
LIN {X 0,Y 65.366,Z 1060.824,A -85,B 0,C 180,E1 4425.072,E2 4425.072} C_VEL
LIN {X 0,Y 64.106,Z 1061.577,A -85,B 0,C 180,E1 4410.894,E2 4410.894} C_VEL
LIN {X 0,Y 64.418,Z 1061.735,A -85,B 0,C 180,E1 4398.358,E2 4398.358} C_VEL
LIN {X 0,Y 67.808,Z 1061.092,A -85,B 0,C 180,E1 4381.844,E2 4381.844} C_VEL
LIN {X 0,Y 75.884,Z 1059.388,A -85,B 0,C 180,E1 4366.75,E2 4366.75} C_VEL
LIN {X 0,Y 90.701,Z 1055.888,A -85,B 0,C 180,E1 4352.696,E2 4352.696} C_VEL
LIN {X 0,Y 107.795,Z 1050.971,A -85,B 0,C 180,E1 4343.319,E2 4343.319} C_VEL
LIN {X 0,Y 128.058,Z 1044.244,A -85,B 0,C 180,E1 4336.179,E2 4336.179} C_VEL
LIN {X 0,Y 148.792,Z 1035.891,A -85,B 0,C 180,E1 4331.148,E2 4331.148} C_VEL
LIN {X 0,Y 169.6,Z 1026.27,A -85,B 0,C 180,E1 4327.453,E2 4327.453} C_VEL
LIN {X 0,Y 190.59,Z 1014.857,A -85,B 0,C 180,E1 4324.587,E2 4324.587} C_VEL
LIN {X 0,Y 210.259,Z 1002.709,A -85,B 0,C 180,E1 4322.453,E2 4322.453} C_VEL
LIN {X 0,Y 230.988,Z 987.939,A -85,B 0,C 180,E1 4320.608,E2 4320.608} C_VEL
LIN {X 0,Y 244.535,Z 977.131,A -85,B 0,C 180,E1 4319.575,E2 4319.575} C_VEL
LIN {X 0,Y 225.092,Z 992.64,A -85,B 0,C 180,E1 4318.152,E2 4318.152} C_VEL
LIN {X 0,Y 205.379,Z 1006.28,A -85,B 0,C 180,E1 4316.415,E2 4316.415} C_VEL
LIN {X 0,Y 184.167,Z 1019.311,A -85,B 0,C 180,E1 4314.079,E2 4314.079} C_VEL
LIN {X 0,Y 162.956,Z 1030.449,A -85,B 0,C 180,E1 4311.074,E2 4311.074} C_VEL
LIN {X 0,Y 141.601,Z 1040.317,A -85,B 0,C 180,E1 4307.023,E2 4307.023} C_VEL
LIN {X 0,Y 129.077,Z 1045.346,A -85,B 0,C 180,E1 4303.936,E2 4303.936} C_VEL
LIN {X 0,Y 122.39,Z 1047.811,A -85,B 0,C 180,E1 4302.53,E2 4302.53} C_VEL
LIN {X 0,Y 102.769,Z 1053.524,A -85,B 0,C 180,E1 4299.544,E2 4299.544} C_VEL
LIN {X 0,Y 97.132,Z 1055.053,A -85,B 0,C 180,E1 4297.701,E2 4297.701} C_VEL
LIN {X 0,Y 78.848,Z 1059.803,A -85,B 0,C 180,E1 4286.821,E2 4286.821} C_VEL
LIN {X 0,Y 65.517,Z 1062.863,A -85,B 0,C 180,E1 4272.184,E2 4272.184} C_VEL
LIN {X 0,Y 57.203,Z 1064.641,A -85,B 0,C 180,E1 4250.462,E2 4250.462} C_VEL
LIN {X 0,Y 56.02,Z 1064.939,A -85,B 0,C 180,E1 4234.094,E2 4234.094} C_VEL
LIN {X 0,Y 56.018,Z 1064.736,A -85,B 0,C 180,E1 4224.88,E2 4224.88} C_VEL
LIN {X 0,Y 57.802,Z 1063.651,A -85,B 0,C 180,E1 4206.465,E2 4206.465} C_VEL
LIN {X 0,Y 67.524,Z 1060.58,A -85,B 0,C 180,E1 4184.701,E2 4184.701} C_VEL
LIN {X 0,Y 81.292,Z 1056.486,A -85,B 0,C 180,E1 4171.104,E2 4171.104} C_VEL
LIN {X 0,Y 101.484,Z 1049.849,A -85,B 0,C 180,E1 4160.172,E2 4160.172} C_VEL
LIN {X 0,Y 120.485,Z 1042.59,A -85,B 0,C 180,E1 4153.841,E2 4153.841} C_VEL
LIN {X 0,Y 142.668,Z 1032.818,A -85,B 0,C 180,E1 4148.812,E2 4148.812} C_VEL
LIN {X 0,Y 162.74,Z 1022.5,A -85,B 0,C 180,E1 4145.533,E2 4145.533} C_VEL
LIN {X 0,Y 184.211,Z 1009.932,A -85,B 0,C 180,E1 4142.871,E2 4142.871} C_VEL
LIN {X 0,Y 204.005,Z 996.526,A -85,B 0,C 180,E1 4140.938,E2 4140.938} C_VEL
LIN {X 0,Y 223.989,Z 981.263,A -85,B 0,C 180,E1 4139.361,E2 4139.361} C_VEL
LIN {X 0,Y 238.066,Z 969.095,A -85,B 0,C 180,E1 4138.399,E2 4138.399} C_VEL
LIN {X 0,Y 218.288,Z 985.57,A -85,B 0,C 180,E1 4136.935,E2 4136.935} C_VEL
LIN {X 0,Y 200.631,Z 998.563,A -85,B 0,C 180,E1 4135.376,E2 4135.376} C_VEL
LIN {X 0,Y 178.323,Z 1012.889,A -85,B 0,C 180,E1 4132.964,E2 4132.964} C_VEL
LIN {X 0,Y 159.241,Z 1023.553,A -85,B 0,C 180,E1 4130.338,E2 4130.338} C_VEL
LIN {X 0,Y 136.887,Z 1034.358,A -85,B 0,C 180,E1 4126.286,E2 4126.286} C_VEL
LIN {X 0,Y 118.037,Z 1042.176,A -85,B 0,C 180,E1 4121.576,E2 4121.576} C_VEL
LIN {X 0,Y 96.962,Z 1049.707,A -85,B 0,C 180,E1 4113.787,E2 4113.787} C_VEL
LIN {X 0,Y 80.417,Z 1054.726,A -85,B 0,C 180,E1 4103.92,E2 4103.92} C_VEL
LIN {X 0,Y 66.011,Z 1058.76,A -85,B 0,C 180,E1 4088.392,E2 4088.392} C_VEL
LIN {X 0,Y 57.807,Z 1060.995,A -85,B 0,C 180,E1 4067.947,E2 4067.947} C_VEL
LIN {X 0,Y 56.124,Z 1061.772,A -85,B 0,C 180,E1 4052.042,E2 4052.042} C_VEL
LIN {X 0,Y 56.368,Z 1061.987,A -85,B 0,C 180,E1 4038.748,E2 4038.748} C_VEL
LIN {X 0,Y 60.39,Z 1061.363,A -85,B 0,C 180,E1 4019.118,E2 4019.118} C_VEL
LIN {X 0,Y 70.121,Z 1059.591,A -85,B 0,C 180,E1 4002.141,E2 4002.141} C_VEL
LIN {X 0,Y 87.01,Z 1055.945,A -85,B 0,C 180,E1 3987.766,E2 3987.766} C_VEL
LIN {X 0,Y 105.641,Z 1050.907,A -85,B 0,C 180,E1 3978.826,E2 3978.826} C_VEL
LIN {X 0,Y 126.912,Z 1044.079,A -85,B 0,C 180,E1 3972.326,E2 3972.326} C_VEL
LIN {X 0,Y 148.361,Z 1035.653,A -85,B 0,C 180,E1 3967.814,E2 3967.814} C_VEL
LIN {X 0,Y 169.517,Z 1026.05,A -85,B 0,C 180,E1 3964.557,E2 3964.557} C_VEL
LIN {X 0,Y 191.095,Z 1014.425,A -85,B 0,C 180,E1 3962,E2 3962} C_VEL
LIN {X 0,Y 211.977,Z 1001.629,A -85,B 0,C 180,E1 3960.046,E2 3960.046} C_VEL
LIN {X 0,Y 216.699,Z 998.359,A -85,B 0,C 180,E1 3959.651,E2 3959.651} C_VEL
LIN {X 0,Y 194.132,Z 1012.942,A -85,B 0,C 180,E1 3957.726,E2 3957.726} C_VEL
LIN {X 0,Y 174.491,Z 1023.956,A -85,B 0,C 180,E1 3955.616,E2 3955.616} C_VEL
LIN {X 0,Y 151.327,Z 1035.224,A -85,B 0,C 180,E1 3952.359,E2 3952.359} C_VEL
LIN {X 0,Y 131.587,Z 1043.397,A -85,B 0,C 180,E1 3948.589,E2 3948.589} C_VEL
LIN {X 0,Y 109.971,Z 1051.117,A -85,B 0,C 180,E1 3942.687,E2 3942.687} C_VEL
LIN {X 0,Y 97.132,Z 1055.053,A -85,B 0,C 180,E1 3937.701,E2 3937.701} C_VEL
LIN {X 0,Y 90.611,Z 1056.71,A -85,B 0,C 180,E1 3935.327,E2 3935.327} C_VEL
LIN {X 0,Y 71.632,Z 1060.475,A -85,B 0,C 180,E1 3929.056,E2 3929.056} C_VEL
LIN {X 0,Y 66.584,Z 1061.353,A -85,B 0,C 180,E1 3925.514,E2 3925.514} C_VEL
LIN {X 0,Y 53.633,Z 1063.713,A -85,B 0,C 180,E1 3906.626,E2 3906.626} C_VEL
LIN {X 0,Y 48.448,Z 1064.62,A -85,B 0,C 180,E1 3885.563,E2 3885.563} C_VEL
LIN {X 0,Y 48.06,Z 1064.66,A -85,B 0,C 180,E1 3871.192,E2 3871.192} C_VEL
LIN {X 0,Y 48.232,Z 1064.311,A -85,B 0,C 180,E1 3856.994,E2 3856.994} C_VEL
LIN {X 0,Y 53.586,Z 1062.502,A -85,B 0,C 180,E1 3833.337,E2 3833.337} C_VEL
LIN {X 0,Y 65.293,Z 1059.487,A -85,B 0,C 180,E1 3815.586,E2 3815.586} C_VEL
LIN {X 0,Y 84.1,Z 1054.308,A -85,B 0,C 180,E1 3801.973,E2 3801.973} C_VEL
LIN {X 0,Y 103.157,Z 1048.11,A -85,B 0,C 180,E1 3794.236,E2 3794.236} C_VEL
LIN {X 0,Y 125.358,Z 1039.722,A -85,B 0,C 180,E1 3788.484,E2 3788.484} C_VEL
LIN {X 0,Y 146.483,Z 1030.188,A -85,B 0,C 180,E1 3784.734,E2 3784.734} C_VEL
LIN {X 0,Y 168.076,Z 1019.049,A -85,B 0,C 180,E1 3781.924,E2 3781.924} C_VEL
LIN {X 0,Y 188.98,Z 1006.39,A -85,B 0,C 180,E1 3779.838,E2 3779.838} C_VEL
LIN {X 0,Y 207.823,Z 993.527,A -85,B 0,C 180,E1 3778.311,E2 3778.311} C_VEL
LIN {X 0,Y 189.285,Z 1006.002,A -85,B 0,C 180,E1 3776.742,E2 3776.742} C_VEL
LIN {X 0,Y 168.439,Z 1018.428,A -85,B 0,C 180,E1 3774.55,E2 3774.55} C_VEL
LIN {X 0,Y 147.516,Z 1029.03,A -85,B 0,C 180,E1 3771.735,E2 3771.735} C_VEL
LIN {X 0,Y 126.765,Z 1038.203,A -85,B 0,C 180,E1 3767.98,E2 3767.98} C_VEL
LIN {X 0,Y 104.937,Z 1046.277,A -85,B 0,C 180,E1 3762.335,E2 3762.335} C_VEL
LIN {X 0,Y 86.145,Z 1052.186,A -85,B 0,C 180,E1 3754.871,E2 3754.871} C_VEL
LIN {X 0,Y 66.651,Z 1057.312,A -85,B 0,C 180,E1 3741.269,E2 3741.269} C_VEL
LIN {X 0,Y 54.829,Z 1060.084,A -85,B 0,C 180,E1 3724.425,E2 3724.425} C_VEL
LIN {X 0,Y 48.729,Z 1061.727,A -85,B 0,C 180,E1 3701.841,E2 3701.841} C_VEL
LIN {X 0,Y 48.068,Z 1062.103,A -85,B 0,C 180,E1 3686.422,E2 3686.422} C_VEL
LIN {X 0,Y 49.156,Z 1062.102,A -85,B 0,C 180,E1 3671.007,E2 3671.007} C_VEL
LIN {X 0,Y 55.293,Z 1061.319,A -85,B 0,C 180,E1 3650.734,E2 3650.734} C_VEL
LIN {X 0,Y 69.814,Z 1058.978,A -85,B 0,C 180,E1 3632,E2 3632} C_VEL
LIN {X 0,Y 88.457,Z 1054.931,A -85,B 0,C 180,E1 3620.248,E2 3620.248} C_VEL
LIN {X 0,Y 109.601,Z 1049.347,A -85,B 0,C 180,E1 3612.536,E2 3612.536} C_VEL
LIN {X 0,Y 131.092,Z 1042.163,A -85,B 0,C 180,E1 3607.449,E2 3607.449} C_VEL
LIN {X 0,Y 152.337,Z 1033.816,A -85,B 0,C 180,E1 3603.904,E2 3603.904} C_VEL
LIN {X 0,Y 175.013,Z 1023.147,A -85,B 0,C 180,E1 3601.092,E2 3601.092} C_VEL
LIN {X 0,Y 188.564,Z 1015.938,A -85,B 0,C 180,E1 3599.703,E2 3599.703} C_VEL
LIN {X 0,Y 165.157,Z 1028.282,A -85,B 0,C 180,E1 3597.36,E2 3597.36} C_VEL
LIN {X 0,Y 144.618,Z 1037.527,A -85,B 0,C 180,E1 3594.632,E2 3594.632} C_VEL
LIN {X 0,Y 121.687,Z 1046.35,A -85,B 0,C 180,E1 3590.41,E2 3590.41} C_VEL
LIN {X 0,Y 100.58,Z 1053.019,A -85,B 0,C 180,E1 3584.645,E2 3584.645} C_VEL
LIN {X 0,Y 79.333,Z 1058.608,A -85,B 0,C 180,E1 3575.158,E2 3575.158} C_VEL
LIN {X 0,Y 66.584,Z 1061.353,A -85,B 0,C 180,E1 3565.514,E2 3565.514} C_VEL
LIN {X 0,Y 60.947,Z 1062.254,A -85,B 0,C 180,E1 3560.774,E2 3560.774} C_VEL
LIN {X 0,Y 48.829,Z 1063.644,A -85,B 0,C 180,E1 3550.398,E2 3550.398} C_VEL
LIN {X 0,Y 43.169,Z 1064.164,A -85,B 0,C 180,E1 3540.881,E2 3540.881} C_VEL
LIN {X 0,Y 42.163,Z 1064.229,A -85,B 0,C 180,E1 3537.388,E2 3537.388} C_VEL
LIN {X 0,Y 40.022,Z 1064.484,A -85,B 0,C 180,E1 3514.299,E2 3514.299} C_VEL
LIN {X 0,Y 40.03,Z 1064.301,A -85,B 0,C 180,E1 3502.826,E2 3502.826} C_VEL
LIN {X 0,Y 44.07,Z 1063.056,A -85,B 0,C 180,E1 3475.444,E2 3475.444} C_VEL
LIN {X 0,Y 57.857,Z 1059.928,A -85,B 0,C 180,E1 3452.133,E2 3452.133} C_VEL
LIN {X 0,Y 74.437,Z 1055.902,A -85,B 0,C 180,E1 3439.901,E2 3439.901} C_VEL
LIN {X 0,Y 97.698,Z 1049.091,A -85,B 0,C 180,E1 3430.731,E2 3430.731} C_VEL
LIN {X 0,Y 117.622,Z 1042.044,A -85,B 0,C 180,E1 3425.957,E2 3425.957} C_VEL
LIN {X 0,Y 141.082,Z 1032.241,A -85,B 0,C 180,E1 3422.131,E2 3422.131} C_VEL
LIN {X 0,Y 160.983,Z 1022.432,A -85,B 0,C 180,E1 3419.785,E2 3419.785} C_VEL
LIN {X 0,Y 177.521,Z 1013.232,A -85,B 0,C 180,E1 3418.248,E2 3418.248} C_VEL
LIN {X 0,Y 158.31,Z 1023.632,A -85,B 0,C 180,E1 3416.313,E2 3416.313} C_VEL
LIN {X 0,Y 134.501,Z 1034.689,A -85,B 0,C 180,E1 3413.169,E2 3413.169} C_VEL
LIN {X 0,Y 114.879,Z 1042.369,A -85,B 0,C 180,E1 3409.589,E2 3409.589} C_VEL
LIN {X 0,Y 92.738,Z 1049.722,A -85,B 0,C 180,E1 3403.654,E2 3403.654} C_VEL
LIN {X 0,Y 72.424,Z 1055.127,A -85,B 0,C 180,E1 3394.66,E2 3394.66} C_VEL
LIN {X 0,Y 54.254,Z 1059.23,A -85,B 0,C 180,E1 3379.08,E2 3379.08} C_VEL
LIN {X 0,Y 42.848,Z 1061.432,A -85,B 0,C 180,E1 3354.837,E2 3354.837} C_VEL
LIN {X 0,Y 40.142,Z 1062.206,A -85,B 0,C 180,E1 3332.855,E2 3332.855} C_VEL
LIN {X 0,Y 40.672,Z 1062.41,A -85,B 0,C 180,E1 3314.31,E2 3314.31} C_VEL
LIN {X 0,Y 47.124,Z 1061.779,A -85,B 0,C 180,E1 3288.87,E2 3288.87} C_VEL
LIN {X 0,Y 60.323,Z 1059.997,A -85,B 0,C 180,E1 3270.465,E2 3270.465} C_VEL
LIN {X 0,Y 80.642,Z 1056.326,A -85,B 0,C 180,E1 3257.305,E2 3257.305} C_VEL
LIN {X 0,Y 100.575,Z 1051.523,A -85,B 0,C 180,E1 3250.19,E2 3250.19} C_VEL
LIN {X 0,Y 123.46,Z 1044.763,A -85,B 0,C 180,E1 3245.018,E2 3245.018} C_VEL
LIN {X 0,Y 146.036,Z 1036.376,A -85,B 0,C 180,E1 3241.525,E2 3241.525} C_VEL
LIN {X 0,Y 160.608,Z 1030.16,A -85,B 0,C 180,E1 3239.804,E2 3239.804} C_VEL
LIN {X 0,Y 137.175,Z 1040.182,A -85,B 0,C 180,E1 3236.981,E2 3236.981} C_VEL
LIN {X 0,Y 114.802,Z 1048.029,A -85,B 0,C 180,E1 3233.172,E2 3233.172} C_VEL
LIN {X 0,Y 92.243,Z 1054.65,A -85,B 0,C 180,E1 3227.311,E2 3227.311} C_VEL
LIN {X 0,Y 71.164,Z 1059.409,A -85,B 0,C 180,E1 3218.024,E2 3218.024} C_VEL
LIN {X 0,Y 53.808,Z 1062.577,A -85,B 0,C 180,E1 3203.04,E2 3203.04} C_VEL
LIN {X 0,Y 42.163,Z 1064.229,A -85,B 0,C 180,E1 3177.388,E2 3177.388} C_VEL
LIN {X 0,Y 39.826,Z 1064.407,A -85,B 0,C 180,E1 3168.669,E2 3168.669} C_VEL
LIN {X 0,Y 36.217,Z 1064.401,A -85,B 0,C 180,E1 3156.276,E2 3156.276} C_VEL
LIN {X 0,Y 33.294,Z 1063.674,A -85,B 0,C 180,E1 3126.035,E2 3126.035} C_VEL
LIN {X 0,Y 33.849,Z 1063.503,A -85,B 0,C 180,E1 3122.236,E2 3122.236} C_VEL
LIN {X 0,Y 43.543,Z 1061.673,A -85,B 0,C 180,E1 3096.513,E2 3096.513} C_VEL
LIN {X 0,Y 62.284,Z 1058.004,A -85,B 0,C 180,E1 3078.708,E2 3078.708} C_VEL
LIN {X 0,Y 84.085,Z 1052.48,A -85,B 0,C 180,E1 3069.253,E2 3069.253} C_VEL
LIN {X 0,Y 107.202,Z 1045.387,A -85,B 0,C 180,E1 3063.622,E2 3063.622} C_VEL
LIN {X 0,Y 130.471,Z 1036.475,A -85,B 0,C 180,E1 3060,E2 3060} C_VEL
LIN {X 0,Y 146.709,Z 1029.307,A -85,B 0,C 180,E1 3058.161,E2 3058.161} C_VEL
LIN {X 0,Y 125.373,Z 1038.359,A -85,B 0,C 180,E1 3055.498,E2 3055.498} C_VEL
LIN {X 0,Y 102.142,Z 1046.505,A -85,B 0,C 180,E1 3051.383,E2 3051.383} C_VEL
LIN {X 0,Y 81.502,Z 1052.448,A -85,B 0,C 180,E1 3045.742,E2 3045.742} C_VEL
LIN {X 0,Y 58.712,Z 1057.638,A -85,B 0,C 180,E1 3034.503,E2 3034.503} C_VEL
LIN {X 0,Y 42.738,Z 1060.505,A -85,B 0,C 180,E1 3017.274,E2 3017.274} C_VEL
LIN {X 0,Y 33.191,Z 1062.175,A -85,B 0,C 180,E1 2987.533,E2 2987.533} C_VEL
LIN {X 0,Y 32.075,Z 1062.519,A -85,B 0,C 180,E1 2965.995,E2 2965.995} C_VEL
LIN {X 0,Y 33.931,Z 1062.547,A -85,B 0,C 180,E1 2943.767,E2 2943.767} C_VEL
LIN {X 0,Y 43.2,Z 1061.799,A -85,B 0,C 180,E1 2918.098,E2 2918.098} C_VEL
LIN {X 0,Y 61.616,Z 1059.549,A -85,B 0,C 180,E1 2899.744,E2 2899.744} C_VEL
LIN {X 0,Y 83.233,Z 1055.513,A -85,B 0,C 180,E1 2889.91,E2 2889.91} C_VEL
LIN {X 0,Y 105.277,Z 1050.216,A -85,B 0,C 180,E1 2884.239,E2 2884.239} C_VEL
LIN {X 0,Y 128.988,Z 1042.849,A -85,B 0,C 180,E1 2880.313,E2 2880.313} C_VEL
LIN {X 0,Y 132.228,Z 1041.722,A -85,B 0,C 180,E1 2879.886,E2 2879.886} C_VEL
LIN {X 0,Y 111.161,Z 1048.78,A -85,B 0,C 180,E1 2876.806,E2 2876.806} C_VEL
LIN {X 0,Y 86.03,Z 1055.529,A -85,B 0,C 180,E1 2871.086,E2 2871.086} C_VEL
LIN {X 0,Y 65.839,Z 1059.71,A -85,B 0,C 180,E1 2863.093,E2 2863.093} C_VEL
LIN {X 0,Y 44.951,Z 1062.924,A -85,B 0,C 180,E1 2845.389,E2 2845.389} C_VEL
LIN {X 0,Y 33.94,Z 1064.111,A -85,B 0,C 180,E1 2818.123,E2 2818.123} C_VEL
LIN {X 0,Y 32.036,Z 1064.238,A -85,B 0,C 180,E1 2792.861,E2 2792.861} C_VEL
LIN {X 0,Y 32.254,Z 1064.005,A -85,B 0,C 180,E1 2775.641,E2 2775.641} C_VEL
LIN {X 0,Y 33.849,Z 1063.503,A -85,B 0,C 180,E1 2762.236,E2 2762.236} C_VEL
LIN {X 0,Y 35.924,Z 1062.949,A -85,B 0,C 180,E1 2749.969,E2 2749.969} C_VEL
LIN {X 0,Y 45.544,Z 1060.543,A -85,B 0,C 180,E1 2721.177,E2 2721.177} C_VEL
LIN {X 0,Y 49.862,Z 1059.662,A -85,B 0,C 180,E1 2717.046,E2 2717.046} C_VEL
LIN {X 0,Y 69.78,Z 1055.57,A -85,B 0,C 180,E1 2707.41,E2 2707.41} C_VEL
LIN {X 0,Y 95.008,Z 1048.871,A -85,B 0,C 180,E1 2701.13,E2 2701.13} C_VEL
LIN {X 0,Y 115.31,Z 1042.129,A -85,B 0,C 180,E1 2698.056,E2 2698.056} C_VEL
LIN {X 0,Y 92.442,Z 1049.426,A -85,B 0,C 180,E1 2694.329,E2 2694.329} C_VEL
LIN {X 0,Y 69.46,Z 1055.115,A -85,B 0,C 180,E1 2688.202,E2 2688.202} C_VEL
LIN {X 0,Y 49.554,Z 1058.954,A -85,B 0,C 180,E1 2678.153,E2 2678.153} C_VEL
LIN {X 0,Y 30.708,Z 1061.689,A -85,B 0,C 180,E1 2653.14,E2 2653.14} C_VEL
LIN {X 0,Y 24.252,Z 1062.618,A -85,B 0,C 180,E1 2617.104,E2 2617.104} C_VEL
LIN {X 0,Y 24.751,Z 1062.878,A -85,B 0,C 180,E1 2591.144,E2 2591.144} C_VEL
LIN {X 0,Y 35.699,Z 1062.259,A -85,B 0,C 180,E1 2552.83,E2 2552.83} C_VEL
LIN {X 0,Y 52.977,Z 1060.511,A -85,B 0,C 180,E1 2535.722,E2 2535.722} C_VEL
LIN {X 0,Y 75.417,Z 1057.108,A -85,B 0,C 180,E1 2526.086,E2 2526.086} C_VEL
LIN {X 0,Y 98.997,Z 1051.89,A -85,B 0,C 180,E1 2520.704,E2 2520.704} C_VEL
LIN {X 0,Y 103.102,Z 1050.871,A -85,B 0,C 180,E1 2519.951,E2 2519.951} C_VEL
LIN {X 0,Y 81.222,Z 1056.191,A -85,B 0,C 180,E1 2515.679,E2 2515.679} C_VEL
LIN {X 0,Y 57.411,Z 1060.608,A -85,B 0,C 180,E1 2507.246,E2 2507.246} C_VEL
LIN {X 0,Y 37.703,Z 1063.012,A -85,B 0,C 180,E1 2491.066,E2 2491.066} C_VEL
LIN {X 0,Y 25.85,Z 1063.981,A -85,B 0,C 180,E1 2460.189,E2 2460.189} C_VEL
LIN {X 0,Y 24.073,Z 1063.988,A -85,B 0,C 180,E1 2430,E2 2430} C_VEL
LIN {X 0,Y 26.511,Z 1063.347,A -85,B 0,C 180,E1 2396.074,E2 2396.074} C_VEL
LIN {X 0,Y 39.216,Z 1061.438,A -85,B 0,C 180,E1 2366.825,E2 2366.825} C_VEL
LIN {X 0,Y 49.862,Z 1059.662,A -85,B 0,C 180,E1 2357.046,E2 2357.046} C_VEL
LIN {X 0,Y 56.048,Z 1058.451,A -85,B 0,C 180,E1 2352.138,E2 2352.138} C_VEL
LIN {X 0,Y 72.979,Z 1054.561,A -85,B 0,C 180,E1 2340.278,E2 2340.278} C_VEL
LIN {X 0,Y 78.535,Z 1053.139,A -85,B 0,C 180,E1 2338.664,E2 2338.664} C_VEL
LIN {X 0,Y 82.675,Z 1052.06,A -85,B 0,C 180,E1 2337.921,E2 2337.921} C_VEL
LIN {X 0,Y 58.551,Z 1057.348,A -85,B 0,C 180,E1 2332.084,E2 2332.084} C_VEL
LIN {X 0,Y 36.185,Z 1060.687,A -85,B 0,C 180,E1 2319.967,E2 2319.967} C_VEL
LIN {X 0,Y 21.273,Z 1062.299,A -85,B 0,C 180,E1 2294.831,E2 2294.831} C_VEL
LIN {X 0,Y 16.14,Z 1062.878,A -85,B 0,C 180,E1 2253.551,E2 2253.551} C_VEL
LIN {X 0,Y 18.509,Z 1063.048,A -85,B 0,C 180,E1 2213.541,E2 2213.541} C_VEL
LIN {X 0,Y 32.871,Z 1062.405,A -85,B 0,C 180,E1 2179.444,E2 2179.444} C_VEL
LIN {X 0,Y 52.324,Z 1060.607,A -85,B 0,C 180,E1 2166.43,E2 2166.43} C_VEL
LIN {X 0,Y 73.451,Z 1057.574,A -85,B 0,C 180,E1 2160.112,E2 2160.112} C_VEL
LIN {X 0,Y 50.122,Z 1061.154,A -85,B 0,C 180,E1 2153.126,E2 2153.126} C_VEL
LIN {X 0,Y 30.141,Z 1063.174,A -85,B 0,C 180,E1 2138.26,E2 2138.26} C_VEL
LIN {X 0,Y 16.511,Z 1063.886,A -85,B 0,C 180,E1 2091.306,E2 2091.306} C_VEL
LIN {X 0,Y 16.029,Z 1063.747,A -85,B 0,C 180,E1 2066.424,E2 2066.424} C_VEL
LIN {X 0,Y 21.014,Z 1063.032,A -85,B 0,C 180,E1 2020.421,E2 2020.421} C_VEL
LIN {X 0,Y 37.164,Z 1061.082,A -85,B 0,C 180,E1 1994.403,E2 1994.403} C_VEL
LIN {X 0,Y 61.062,Z 1057.076,A -85,B 0,C 180,E1 1982.727,E2 1982.727} C_VEL
LIN {X 0,Y 78.535,Z 1053.139,A -85,B 0,C 180,E1 1978.664,E2 1978.664} C_VEL
LIN {X 0,Y 76.858,Z 1053.554,A -85,B 0,C 180,E1 1977.954,E2 1977.954} C_VEL
LIN {X 0,Y 67.643,Z 1055.539,A -85,B 0,C 180,E1 1977.385,E2 1977.385} C_VEL
LIN {X 0,Y 48.871,Z 1059.025,A -85,B 0,C 180,E1 1978.414,E2 1978.414} C_VEL
LIN {X 0,Y 36.149,Z 1060.829,A -85,B 0,C 180,E1 1981.559,E2 1981.559} C_VEL
LIN {X 0,Y 16.908,Z 1062.805,A -85,B 0,C 180,E1 1998.88,E2 1998.88} C_VEL
LIN {X 0,Y 8.025,Z 1063.538,A -85,B 0,C 180,E1 2065.359,E2 2065.359} C_VEL
LIN {X 0,Y 13.539,Z 1063.581,A -85,B 0,C 180,E1 2132.405,E2 2132.405} C_VEL
LIN {X 0,Y 32.306,Z 1062.649,A -85,B 0,C 180,E1 2156.451,E2 2156.451} C_VEL
LIN {X 0,Y 41.628,Z 1061.928,A -85,B 0,C 180,E1 2160.32,E2 2160.32} C_VEL
LIN {X 0,Y 18.822,Z 1063.133,A -85,B 0,C 180,E1 2177.017,E2 2177.017} C_VEL
LIN {X 0,Y 8.44,Z 1063.189,A -85,B 0,C 180,E1 2229.18,E2 2229.18} C_VEL
LIN {X 0,Y 10.496,Z 1062.969,A -85,B 0,C 180,E1 2291.823,E2 2291.823} C_VEL
LIN {X 0,Y 29.443,Z 1061.463,A -85,B 0,C 180,E1 2330.015,E2 2330.015} C_VEL
LIN {X 0,Y 47.59,Z 1059.195,A -85,B 0,C 180,E1 2337.763,E2 2337.763} C_VEL
LIN {X 0,Y 36.149,Z 1060.829,A -85,B 0,C 180,E1 2341.559,E2 2341.559} C_VEL
LIN {X 0,Y 26.677,Z 1061.947,A -85,B 0,C 180,E1 2344.819,E2 2344.819} C_VEL
LIN {X 0,Y 13.532,Z 1062.899,A -85,B 0,C 180,E1 2346.932,E2 2346.932} C_VEL
LIN {X 0,Y 0.342,Z 1063.344,A -85,B 0,C 180,E1 2520.312,E2 2520.312} C_VEL
LIN {X 0,Y 0.649,Z 1063.35,A -85,B 0,C 180,E1 2523.034,E2 2523.034} C_VEL
LIN {X 0,Y 1.003,Z 1063.312,A -85,B 0,C 180,E1 2695.574,E2 2695.574} C_VEL
LIN {X 0,Y 0.342,Z 1063.344,A -85,B 0,C 180,E1 2520.312,E2 2520.312} C_VEL
LIN {X 0,Y 2.302,Z 1065.344,A -85,B 0,C 180,E1 2525.206,E2 2525.206} C_VEL
LIN {X 0,Y 2.302,Z 1088.5,A -85,B 0,C 180,E1 2525.206,E2 2525.206} C_VEL
LIN {X 0,Y 2.302,Z 1088.5,A -85,B 0,C 180,E1 2525.206,E2 2525.206}

QRS_NEXT_CUT()

QRS_NEXT()
QRS_HOME()

END
